(* RESETS AXES IF PHASE DONE AND CONNECTION DONE AND DISABLED *)
IF 	phase_done
	AND connection_done
	AND axis_is_disabled(axis)
THEN
	phase_done := FALSE;
	connection_done := FALSE;
END_IF

(* CLEARS PHASE AND CONNECTION ERRORS ON STOP *)
IF 	machine_is_stopped(csp.mch)
	OR machine_is_stop_emergency_active(csp.mch)
THEN
	phase_error := FALSE;
	connection_error := FALSE;	
END_IF

(* Overflow protection of engage count *)
IF	engage_count > 32000
THEN
	engage_count := 0;
END_IF

phase();

connection();

_handle_messages();

_write_output();

ACTION _handle_messages:
;
END_ACTION

ACTION _handle_process_test:
;
END_ACTION

ACTION _mode_manager:
IF process_mode_req_is_pending(prc)
THEN
    process_apply_mode_req_first_step(prc);
    CASE process_get_mode(prc) OF
        MODE_TO_ABSENT:
			;
        MODE_TO_INACTIVE:
			;
        MODE_TO_TEST:
			;
        MODE_TO_OPERATIONAL:
			;
    END_CASE
    process_apply_mode_req_second_step(prc);
END_IF
END_ACTION

ACTION _object_manager:
IF objects_initialization()
THEN
	sub_process_init(
		object_name					:= 'csp_case_virtualMaster.prc', 
		process						:= csp_case.prc, 
		CONVERSION_this				:= prc);
		
	prc_path 						:= process_get_path(prc);
	
	boolean_init(
        object_name:= CONCAT(prc_path, 'Axis_faulted'),
        process:= prc,
        CONVERSION_this:= Axis_faulted);
		
	axis_init(
		object_name								:= CONCAT(prc_path, '_axis'), 
		axis_type								:= AXIS_TYPE_VIRTUAL, 
		encoder_scaling_factor					:= G_VIRTUAL_ENCODER_SCALING_FACTOR_DEGPINC,
		modulo									:= G_MODULO_360_DEG, 
		process									:= prc, 
		CONVERSION_this							:= axis);
	
	axis_set_max_dynamic(
		reference_velocity						:=	MOTOR_MAX_VELOCITY_DEGPS,
		velocity								:=	MOTOR_MAX_VELOCITY_DEGPS,
		acceleration							:=	MOTOR_MAX_ACCELLERATION_DEGPS2,
		deceleration							:=	MOTOR_MAX_DECELLERATION_DEGPS2,
		jerk									:=	MOTOR_MAX_JERK_DEGPS3,
		following_error							:=	MOTOR_MAX_FOLLOWING_ERROR_DEG,
		CONVERSION_this							:=	axis);
	
	jog_manager_add_axis(
		list_index					:= JOG_LIST_CSP_CASE_VIRTUAL,
		axis						:= axis,
		master_axis					:= TRUE,
		jog_type					:= JOG_TYPE_ROTATIVE_PLUS,
		sw_limit_positive			:= 0.0,
		sw_limit_negative			:= 0.0,
		CONVERSION_this				:= csp_main_jogManager.jog_manager_virtual);

	
    digital_check_and_message_init(
        object_name:= CONCAT(prc_path, 'Axis_faulted_active_dchk'),
        alarm_if_input_off:= FALSE,
        alarm_delay:= 0,
        enabled_at_powerup:= TRUE,
        individual_reset:= FALSE,
        machine_reaction:=  MACHINE_REACTION_EMERGENCY_STOP,//MACHINE_REACTION_EMERGENCY_STOP,
        typology:=  MESSAGE_TYPOLOGY_ABNORMAL,//MESSAGE_TYPOLOGY_OBLIGATION,
        process:= prc,
        CONVERSION_this:= Axis_faulted_active_dchk);
       
       
    digital_check_add_boolean(
        boolean:= Axis_faulted,
        CONVERSION_this:= Axis_faulted_active_dchk);

		
	process_message_init(
		object_name					:=	CONCAT(prc_path, '_runout_complete'), 
		behaviour					:=	MESSAGE_BEHAVIOUR_EVENT,
		reset_timeout				:=	0,
		disableable					:=	TRUE,
		individual_reset			:=	FALSE,
		machine_reaction			:=	MACHINE_REACTION_STOP_IN_PHASE_ONE,
		typology					:=	MESSAGE_TYPOLOGY_ABNORMAL,
		process						:=	prc,
		CONVERSION_this				:=	runout_complete);
		
		
	process_message_init(
		object_name					:=	CONCAT(prc_path, '_phase_faulted_aem'), 
		behaviour					:=	MESSAGE_BEHAVIOUR_EVENT,
		reset_timeout				:=	0,
		disableable					:=	TRUE,
		individual_reset			:=	FALSE,
		machine_reaction			:=	MACHINE_REACTION_NORMAL_STOP,
		typology					:=	MESSAGE_TYPOLOGY_ABNORMAL,
		process						:=	prc,
		CONVERSION_this				:=	phase_faulted_aem);
	
	timer_init(
		object_name					:= CONCAT(prc_path, 'phase_time_out_tmr'),
		process						:= prc,
		CONVERSION_this				:= phase_time_out_tmr);
		
	process_message_init(
		object_name					:=	CONCAT(prc_path, 'debug_immediate_stop_aem'), 
		behaviour					:=	MESSAGE_BEHAVIOUR_STATE,
		reset_timeout				:=	0,
		disableable					:=	TRUE,
		individual_reset			:=	FALSE,
		machine_reaction			:=	MACHINE_REACTION_NORMAL_STOP,
		typology					:=	MESSAGE_TYPOLOGY_ABNORMAL,
		process						:=	prc,
		CONVERSION_this				:=	debug_immediate_stop_aem);
		
	timer_init(
		object_name					:= CONCAT(prc_path, 'connection_time_out_tmr'),
		process						:= prc,
		CONVERSION_this				:= connection_time_out_tmr);
		
		
	process_message_init(
		object_name					:=	CONCAT(prc_path, '_connection_faulted_aem'), 
		behaviour					:=	MESSAGE_BEHAVIOUR_EVENT,
		reset_timeout				:=	0,
		disableable					:=	TRUE,
		individual_reset			:=	FALSE,
		machine_reaction			:=	MACHINE_REACTION_NORMAL_STOP,
		typology					:=	MESSAGE_TYPOLOGY_ABNORMAL,
		process						:=	prc,
		CONVERSION_this				:=	connection_faulted_aem);
		
	motorization_conditioner_init(
		object_name					:=	CONCAT(prc_path, 'connection_done_motcond'),
		velocity_limit				:=	0.0,
		velocity_limit_active		:=	FALSE,
		idle_handshake_active		:=	FALSE,
		execute_handshake_active	:=	TRUE,
		hold_handshake_active		:=	FALSE,
		suspend_handshake_active	:=	FALSE,
		complete_handshake_active	:=	FALSE,
		abort_handshake_active		:=	FALSE,
		stop_handshake_active		:=	FALSE,
		origin						:=	MOTORIZATION_CONDITIONER_ORIGIN_INTERNAL,
		manager						:=	csp_main_motorization_manager.motm,
		process						:=	prc,
		CONVERSION_this				:=	connection_done_motcond);
   
		
	phase_init(
        object_name 				:= CONCAT(prc_path, '_run_check_ph'),
        phase 						:= 0,	//Set at runtime!
        delay 						:= 0,
        max_compensation 			:= 0,
        generator 					:= csp_main_motorization_virtualManager.phgen,
        process 					:= prc,
        CONVERSION_this 			:= run_check_ph);	
		
	phase_init(
        object_name 				:= CONCAT(prc_path, '_load_check_ph_jog'),
        phase 						:= 0,	//Set at runtime!
        delay 						:= 0,
        max_compensation 			:= 0,
        generator 					:= csp_main_motorization_virtualManager.phgen,
        process 					:= prc,
        CONVERSION_this 			:= load_check_ph_jog);	
		

END_IF

IF objects_running()
THEN
	process_cycle(prc);
	motorization_conditioner_cycle(connection_done_motcond);
	
	phase_cycle(run_check_ph);
	phase_cycle(load_check_ph_jog);
	axis_cycle(axis);
	digital_check_cycle(Axis_faulted_active_dchk);
END_IF
END_ACTION

ACTION _read_process_image:
;
END_ACTION

ACTION _read_var_input:
disable_req := csp_case.disable_req;
END_ACTION

ACTION _set_runtime_properties:
(* Cam management *)
IF 	connection_done
THEN
	active_cam := axis.engaged_cam.cam_id;
END_IF

(******************** DEBUG *****************************)

IF 
( (* USED FOR PRIMING THE CASE SIDE WITH A CASE SO IT IS READY TO LOAD IMMEDIATELY FROM TRANSFER *)
	(
		NOT csp_case_loader.cases_primed 
		AND 
			(
				NOT csp_case_loader.case_at_loader
				OR
				(
					csp_case_loader.case_at_loader
					AND csp_transfer_upstacker.stack_in_case_at_loader
				)
					
			)
	)
	AND NOT csp_case_transport_virtualMaster.stop_for_reject
	AND axis_is_cam_engaged(csp_case_feed_virtualMaster.axis)
	AND NOT message_is_on(csp_case_discharge_reject_sensors.downstream_backup_di_dchk.alarm_asm.message)
	AND NOT message_is_on(csp_main_interface.Cartoner_Stop_Request_aem)
	AND NOT motorization_manager_is_held(csp_main_motorization_manager.motm)//message_is_on(csp_main_interface.Cartoner_Stop_Request_aem)
	//AND NOT csp_case_feed_magazine.suspend_request_aml_zone	
)
THEN
	condition1 := TRUE;
ELSE
	condition1 := FALSE;
END_IF

IF
( (* STACK IS READY AND WAITING ON TRANSFER TO RUN (CASE & LOAD AT LOAD SR STEP AND CASE AT FEED SR STEP)*)
	csp_case_loader.case_at_loader
	AND csp_transfer_upstacker.stack_in_case_at_loader
	AND csp_case_loader.cases_primed 
	AND csp_case_fc_ls_upper_leadingMinorCloser.at_upstream_pos
	AND NOT csp_case_transport_virtualMaster.stop_for_reject
	AND axis_is_cam_engaged(csp_case_feed_virtualMaster.axis)
	AND axis_is_cam_engaged(csp_case_transport_virtualMaster.axis)
	AND NOT message_is_on(csp_case_discharge_reject_sensors.downstream_backup_di_dchk.alarm_asm.message)
	AND NOT message_is_on(csp_main_interface.Cartoner_Stop_Request_aem)
	AND NOT motorization_manager_is_held(csp_main_motorization_manager.motm)
	//AND NOT csp_case_feed_magazine.suspend_request_aml_zone	
)
THEN
	condition2 := TRUE;
ELSE
	condition2 := FALSE;
END_IF

IF 
( (* STACK IS READY AND WAITING ON TRANSFER TO RUN (NO CASE & LOAD AT LOAD SR STEP AND CASE AT FEED SR STEP) *)
	NOT csp_case_loader.case_at_loader
	AND NOT csp_transfer_upstacker.stack_in_case_at_loader
	AND csp_case_loader.cases_primed 
	//AND NOT csp_case_fc_ls_upper_leadingMinorCloser.at_upstream_pos  //removed because no case at loader
	AND NOT csp_case_transport_virtualMaster.stop_for_reject
	AND axis_is_cam_engaged(csp_case_feed_virtualMaster.axis)
	AND axis_is_cam_engaged(csp_case_transport_virtualMaster.axis)
	AND NOT message_is_on(csp_case_discharge_reject_sensors.downstream_backup_di_dchk.alarm_asm.message)
	AND NOT message_is_on(csp_main_interface.Cartoner_Stop_Request_aem)
	AND NOT motorization_manager_is_held(csp_main_motorization_manager.motm)//message_is_on(csp_main_interface.Cartoner_Stop_Request_aem)
	//AND NOT csp_case_feed_magazine.suspend_request_aml_zone	
	)
THEN
	condition3 := TRUE;
ELSE
	condition3 := FALSE;
END_IF
END_ACTION

ACTION _write_output:
;
END_ACTION

ACTION connection:
connection_conditions :=	
	NOT process_message_is_on(connection_faulted_aem)
	//AND
	//NOT jog_manager_is_jog_axis_active(JOG_LIST_CSP_CASE_VIRTUAL, csp_main_jogManager.jog_manager_virtual)
	AND
	phase_done;

(* connection_done reset *)
IF	connection_done
	AND	
	NOT connection_conditions
	AND
	NOT csp.o_machine_is_running
THEN
	connection_done := FALSE;
END_IF

(* Exit conditions *)
IF	NOT connection_conditions 
	AND
	NOT motorization_manager_is_stopping(csp_main_motorization_manager.motm)	
THEN	
	connection_status_next := CSP_CASE_STATUS_CONNECTION_ERROR;
	connection_status := connection_status_next;	
END_IF

(*************** MACHINE STATUS ***************)
CASE connection_status OF

	CSP_CASE_STATUS_CONNECTION_START:	(* Start connection *)
		IF	(
				motorization_manager_is_starting(csp_main_motorization_manager.motm) //TODOPZ: da decidere a che livello usare le variabili di i e o: wn_feeding.i_motorization_is_starting?					
				//AND axis_is_cam_engaged(csp_case_feed_virtualMaster.axis)
				//AND axis_is_cam_engaged(csp_case_glue_virtualMaster.axis)
				AND 
					(
						axis_is_cam_engaged(csp_case_transport_virtualMaster.axis) 
						OR 
						csp_case_transport_virtualMaster.stop_for_reject
					)
				//AND axis_is_cam_engaged(csp_case_loader_virtualMaster.axis)
				//OR
				//jog_manager_is_jog_axis_active(JOG_LIST_CSP_CASE_VIRTUAL, csp_main_jogManager.jog_manager_virtual)
			)
			THEN
				connection_running := TRUE;
				connection_status_next := CSP_CASE_STATUS_CONNECTION_ENGAGE;
		END_IF
		
	CSP_CASE_STATUS_CONNECTION_ENGAGE:		
	
		master_offset_phase := csp_main_motorization_virtualManager.axis.actual_modulo_position;		
	
		axis_engage_cam(
			cam_id							:=	active_cam,	
			master_engage_mode				:=	AXIS_CAM_ENGAGE_RELATIVE,
			slave_engage_mode				:=	AXIS_CAM_ENGAGE_RELATIVE,
			activation_mode					:=	AXIS_CAM_ACTIVATION_IMMEDIATELY,
			activation_position				:=	0.0,
			master_scaling_mode				:=	AXIS_CAM_SCALING_MODE_USER_DEFINED,
			slave_scaling_mode				:=	AXIS_CAM_SCALING_MODE_AUTOOFFSET,
			master_offset					:=	LMOD(home_position_master_offset_deg + master_offset_phase, axis_get_modulo(csp_main_motorization_virtualManager.axis)),
			slave_offset					:=	0.0,
			master_scaling					:=	master_scaling,
			slave_scaling					:=	slave_scaling,
			interpolation_type				:=	AXIS_CAM_INTERPOLATION_SPLINE,	 
			master							:=	csp_main_motorization_virtualManager.axis,
			CONVERSION_this					:=	axis);
		
		connection_status_next:= CSP_CASE_STATUS_CONNECTION_ENGAGED;
	
	CSP_CASE_STATUS_CONNECTION_ENGAGED:
	
		IF active_cam = 0
		THEN
			active_cam := next_cam;
		END_IF
	
		IF 	axis_is_cam_engaged(axis) 
		THEN				
			IF	active_cam <> next_cam
			THEN							
				connection_status_next := CSP_CASE_STATUS_CONNECTION_CHANGE_CAM;
			ELSE
				connection_status_next:= CSP_CASE_STATUS_CONNECTION_DONE;
			END_IF
		END_IF
		
	CSP_CASE_STATUS_CONNECTION_CHECK_CHANGE_CAM:	
					
		IF 	dwell
		THEN
			next_cam := DWELL_CAM;
			dwell:= FALSE;	
		END_IF
				
		IF 	run
		THEN
			next_cam := FORWARD_CAM;
			run := FALSE;
		END_IF	
		
		IF	(active_cam <> next_cam)
			AND 
			connection_conditions
		THEN							
			connection_status_next := CSP_CASE_STATUS_CONNECTION_CHANGE_CAM;
		END_IF
			
		//IF	NOT connection_motorization_moving
		//THEN
			//connection_status_next := CSP_CASE_STATUS_CONNECTION_DONE;
		//END_IF
	
	CSP_CASE_STATUS_CONNECTION_CHANGE_CAM:	
		engage_count := engage_count + 1;

		axis_engage_cam(
			cam_id							:=	next_cam,	
			master_engage_mode				:=	AXIS_CAM_ENGAGE_RELATIVE,
			slave_engage_mode				:=	AXIS_CAM_ENGAGE_RELATIVE,
			activation_mode					:=	AXIS_CAM_ACTIVATION_NEXT_CYCLE,
			activation_position				:=	0,
			master_scaling_mode				:=	AXIS_CAM_SCALING_MODE_USER_DEFINED,
			slave_scaling_mode				:=	AXIS_CAM_SCALING_MODE_USER_DEFINED,
			master_offset					:=	home_position_master_offset_deg, 
			slave_offset					:=	0.0,
			master_scaling					:=	master_scaling,
			slave_scaling					:=	slave_scaling,
			interpolation_type				:=	AXIS_CAM_INTERPOLATION_SPLINE,	 
			master							:=	csp_main_motorization_virtualManager.axis,
			CONVERSION_this					:=	axis);	
	
		IF	motorization_manager_is_starting(csp_main_motorization_manager.motm)
		THEN
			connection_status_next := CSP_CASE_STATUS_CONNECTION_DONE;
		ELSE
			//IF axis_is_cam_engaged(axis)
			//THEN
			connection_status_next := CSP_CASE_STATUS_CONNECTION_WAIT_NEW_CAM;
		END_IF
		//END_IF
	
	CSP_CASE_STATUS_CONNECTION_WAIT_NEW_CAM:
	
		IF	NOT connection_motorization_moving
		THEN
			connection_status_next := CSP_CASE_STATUS_CONNECTION_DONE;
		END_IF
	
		IF	active_cam = next_cam
		THEN
			connection_status_next := CSP_CASE_STATUS_CONNECTION_CHECK_CHANGE_CAM;
		END_IF
		
	CSP_CASE_STATUS_CONNECTION_DONE:	(* Connection done *)	
	
		connection_running := FALSE;
		connection_done := TRUE;
		
		IF	motorization_manager_is_starting(csp_main_motorization_manager.motm)
		THEN
			motorization_conditioner_start_done(connection_done_motcond);							
			//IF	active_cam <> next_cam
			//THEN
				//connection_status_next := CSP_CASE_STATUS_CONNECTION_WAIT_NEW_CAM;
			//ELSE
				
			//END_IF
		END_IF
		
		IF csp.o_machine_is_running 
		THEN
			connection_status_next := CSP_CASE_STATUS_CONNECTION_CHECK_CHANGE_CAM;
		ELSE
			;//DO NOTHING!! NO NEED TO RUN WHILE NOT IN EXECUTE
		END_IF
	
	CSP_CASE_STATUS_CONNECTION_ERROR:	(* Connection error *)	
	
		IF 	connection_running
		THEN
			axis_disable(axis);
			connection_error := TRUE;						
		END_IF
		connection_running	:= FALSE;
		connection_done 	:= FALSE;	
		
		IF	connection_conditions
		THEN		
			connection_status_next := CSP_CASE_STATUS_CONNECTION_START;
		END_IF
		
END_CASE

IF 	NOT debug_state_machine
	OR
	debug_connection_machine_one_step	
THEN
	connection_status := connection_status_next;
	debug_connection_machine_one_step := FALSE;
END_IF

connection_motorization_moving	:= 
	motorization_manager_is_starting(csp_main_motorization_manager.motm)
	OR
	motorization_manager_is_execute(csp_main_motorization_manager.motm)
	OR
	motorization_manager_is_stopping(csp_main_motorization_manager.motm)
	OR
	motorization_manager_is_suspended(csp_main_motorization_manager.motm)
	OR
	motorization_manager_is_suspending(csp_main_motorization_manager.motm)
	OR
	motorization_manager_is_unsuspending(csp_main_motorization_manager.motm)
	OR 
	motorization_manager_is_holding(csp_main_motorization_manager.motm)
	OR
	motorization_manager_is_held(csp_main_motorization_manager.motm)
	OR
	motorization_manager_is_unholding(csp_main_motorization_manager.motm);	
	
(* Connection timeout *)
IF	(connection_running
	AND NOT debug_state_machine)	
	OR connection_error
THEN
	IF	timer_is_expired(connection_time_out_tmr)
	THEN
		process_message_set(1, connection_status, 0, connection_faulted_aem);
	END_IF
ELSE
	timer_restart(10000, connection_time_out_tmr);
END_IF
END_ACTION

ACTION phase:
phase_conditions :=
	axis_is_ok(FALSE, axis)
	AND
	process_is_ready(prc)
	AND
	process_subtree_is_ready(prc)
	AND
	NOT jog_manager_is_jog_axis_active(JOG_LIST_CSP_CASE_VIRTUAL, csp_main_jogManager.jog_manager_virtual)
	AND
	csp_main_motorization.motorization_axis_redefined_at_powerup
	AND
	NOT disable_req;		
	
(* phase_done reset *)
IF	phase_done
	AND
	NOT phase_conditions
	//AND 
	//NOT csp.o_machine_is_running
THEN
	//axis_disable(axis);
	phase_done:= FALSE;
END_IF

(* Exit condition *)
IF 	NOT phase_conditions
THEN
	phase_status_next := CSP_CASE_PHASE_STATUS_ERROR;
	phase_status := phase_status_next;	
END_IF

(*************** MACHINE STATUS ***************)
CASE phase_status OF

	CSP_CASE_PHASE_STATUS_START:	(* Start phasing *)
	
		IF	(
				motorization_manager_is_starting(csp_main_motorization_manager.motm) //TODOPZ: da decidere a che livello usare le variabili di i e o: wn_feeding.i_motorization_is_starting?					
				//OR
				//jog_manager_is_jog_axis_active(JOG_LIST_CSP_CASE_VIRTUAL, csp_main_jogManager.jog_manager_virtual)
			)
		THEN
			phase_running := TRUE;			
			phase_status_next := CSP_CASE_PHASE_STATUS_DISABLE;
		END_IF
						
	CSP_CASE_PHASE_STATUS_DISABLE:
	
		axis_disable(axis);		
		
		IF 	axis_is_disabled(axis)
		THEN
			phase_status_next := CSP_CASE_PHASE_STATUS_ENABLE;
		END_IF
		
	CSP_CASE_PHASE_STATUS_ENABLE:
	
		axis_enable(axis);
		
		IF 	axis_is_enabled(axis)
		THEN
			phase_status_next := CSP_CASE_PHASE_STATUS_ENABLED;
		END_IF
		
	CSP_CASE_PHASE_STATUS_ENABLED:
	
		IF 	axis_is_standstill(axis) 
		THEN
			phase_status_next := CSP_CASE_PHASE_STATUS_CALCULATE_SLAVE_POSITION_REQUEST;								
		END_IF
		
	CSP_CASE_PHASE_STATUS_CALCULATE_SLAVE_POSITION_REQUEST:
	
		slave_position_has_been_calculated := FALSE;
	
		(* Gets the position of the master axis *)
		axis_calculate_cam_slave_master_position_deg := 
			LMOD(axis_get_actual_modulo_position(csp_main_motorization_virtualManager.axis)
			+ home_position_master_offset_deg, G_MODULO_360_DEG);
			
		(* Gets cam data for slave axis to master *)
		IF 	axis_calculate_cam_slave_dynamics_data(
				cam_id := active_cam,
				master_scaling := master_scaling,
				master_position := axis_calculate_cam_slave_master_position_deg,
				slave_scaling := slave_scaling,
				CONVERSION_this := axis)
		THEN
			phase_status_next := CSP_CASE_PHASE_STATUS_CALCULATING_SLAVE_POSITION;
		END_IF
	
	CSP_CASE_PHASE_STATUS_CALCULATING_SLAVE_POSITION:
	
		IF 	axis_cam_slave_dynamics_data_calculated(axis)
		THEN
			axis_calculated_cam_slave_position_deg := axis_get_cam_slave_dynamics_position(axis);
			slave_position_has_been_calculated := TRUE;
			phase_status_next := CSP_CASE_PHASE_STATUS_REQUEST;
		END_IF
		
	CSP_CASE_PHASE_STATUS_REQUEST:
		
		IF	axis_is_standstill(axis)
		THEN
		 	axis_move_absolute(
				position 		:= axis_calculated_cam_slave_position_deg,
				velocity 		:= phase_velocity_degps,
				direction		:= AXIS_SHORTEST_WAY,
				acceleration 	:= MOTOR_MAX_ACCELLERATION_DEGPS2,
				deceleration 	:= MOTOR_MAX_DECELLERATION_DEGPS2, 
				jerk 			:= MOTOR_MAX_JERK_DEGPS3, 
				buffer_mode 	:= AXIS_BUFFER_MODE_BUFFERED,
				CONVERSION_this := axis
				); 
			
		END_IF

		IF 	axis_is_absolute_moving(axis)
		THEN
			phase_status_next	:=	CSP_CASE_PHASE_STATUS_PHASING;
		END_IF

	CSP_CASE_PHASE_STATUS_PHASING:

		IF 	axis_is_standstill(axis)
		THEN
			phase_status_next	:=	CSP_TRANSFER_STATUS_PHASED;
		END_IF

	CSP_TRANSFER_STATUS_PHASED:

		IF 	engage_enable
		THEN
			phase_status_next := CSP_CASE_PHASE_STATUS_DONE;
		END_IF
		
		
	CSP_CASE_PHASE_STATUS_DONE:	(* Phase done *)		
	
		phase_running := FALSE;
		phase_done := TRUE;				
	
	CSP_CASE_PHASE_STATUS_ERROR:	(* Phase error *)
		

		IF	phase_running
		THEN
			phase_error := TRUE;
			axis_disable(axis);									
		END_IF
		phase_running := FALSE;
		
		IF	phase_conditions 	
		THEN
			phase_status_next := CSP_CASE_PHASE_STATUS_START;
		END_IF
		
END_CASE

IF 	NOT debug_state_machine
	OR
	debug_phase_machine_one_step	
THEN
	phase_status := phase_status_next;
	debug_phase_machine_one_step := FALSE;
END_IF

(* Phasing timeout *)
IF (phase_running
	AND NOT debug_state_machine)
	OR phase_error
THEN
	IF	timer_is_expired(phase_time_out_tmr)
	THEN
		process_message_set(1, phase_status, 0, phase_faulted_aem);
	END_IF
ELSE
	timer_restart(10000, phase_time_out_tmr);
END_IF
END_ACTION

END_PROGRAM

// ---- Application/CSP/Case/Loader/Pusher/csp_case_loader_pusher.TcPOU
(*********************************** G.D S.p.A. - Technical Department ***********************************
============= PROGRAM INFO ============
FOLDER:             TBD
MACHINES INVOLVED:  TBD 

============= DESCRIPTION =============
csp machine declaration

============= REVISIONS ===============
Date		Version	 	Author      	Description             
----------	-------		------------  	--------------------------------------------
2019/04/05 	0000.00	 	M.Grasso		Creation of the PRG

**********************************************************************************************************)
(*$R process_ref := prc; $*)
PROGRAM csp_case_loader_pusher
VAR
	
	prc:											process;
	prc_path:										STRING;
	
	axis:											axis;
	
	fsm_next_status: 								CSP_CASE_LOADER_STATUS_ENUM;
	axis_calculate_cam_slave_master_position_deg: 	LREAL;
	axis_calculated_cam_slave_position_deg: 		LREAL;
	cam_id:											INT := CASE_LOADER_PUSHER_RUN_CAM;
	slave_scaling:									LREAL := 807; (*$P $*) //orginally 360
	master_scaling:									LREAL := 1; 
	master_offset:									LREAL := 240;(*$P $*)
	slave_offset: 									LREAL := 0;
	debug_state_machine: 							BOOL :=FALSE;
	debug_state_machine_one_step: 					BOOL := FALSE;
	fsm_status: 									CSP_CASE_LOADER_STATUS_ENUM;
	phase_velocity_degps: 							LREAL := 50;
	slave_position_has_been_calculated: 			BOOL := FALSE;
	fsm_enable_condition: 							BOOL := FALSE;
	disable_req: 									BOOL := FALSE;
	phase_enable:									BOOL:=TRUE;
	torque_limit:									INT := 2000;    (*$P $*)
	torque_limit_old:								INT;
	
    in_accu_safe_pos:                               BOOL := FALSE;
    accu_tolerance:                                 LREAL := 5;
    accu_safe_pos:                                  LREAL := 0;	
	
	direction_FWD: 									BOOL;
	CAM_CHANGE_CHECK_DEG:							LREAL := 5;
	cam_change_check_ph:							phase;
	
	
	(* RFID *)
	rfid_check_pos:									LREAL := 0; (*$P $*)
	check_pls_tolerance:							LREAL := 2;
	rfid_value:										BYTE;
	rfid_value_to_write:							BYTE;
	
	rfid_input_buffer:								iol_slave_bis00lh_pdo_input;
	rfid_input_bitheader_1:							iol_slave_bis00lh_bitheader_input;
	rfid_input_bitheader_2:							iol_slave_bis00lh_bitheader_input;
			
	rfid_output_buffer:								iol_slave_bis00lh_pdo_output;
	rfid_output_bitheader_1:						iol_slave_bis00lh_bitheader_output;
	rfid_output_bitheader_2:						iol_slave_bis00lh_bitheader_output;
	
	RFID_read_write_status:							csp_case_loader_rfid_status_enum;
	RFID_read_write_status_next:					csp_case_loader_rfid_status_enum;
	RFID_read_write_debug:							BOOL := FALSE;
	RFID_read_write_one_step:						BOOL := FALSE;
	RFID_read_write_running:						BOOL;
	RFID_read_write_tmr:							timer;
	RFID_read_write_error_msg:						message;
	
	rfid_start_toggle:								BOOL := FALSE;
	rfid_shutdown_toggle:							BOOL := FALSE;
	rfid_write_toggle:								BOOL := FALSE;
	rfid_write_done:								BOOL := FALSE;
	rfid_read_toggle:								BOOL := FALSE;
	rfid_read_done:									BOOL := FALSE;

	servo_on_condition: 							BOOL;
	enable_delay: 									TON;
	Torque_force_constant: 							LREAL := 1.2;
	RisingEdgeRFIDSelect:							R_Trig;
END_VAR

VAR CONSTANT
	(*Just in case you prefer having constants instead of numbers*)
	MOTOR_MAX_VELOCITY_DEGPS:				LREAL := 9600;
	MOTOR_MAX_ACCELLERATION_DEGPS2:			LREAL := 4800;
	MOTOR_MAX_DECELLERATION_DEGPS2:			LREAL := 4800;
	MOTOR_MAX_JERK_DEGPS3:					LREAL := 100000000; 
	MOTOR_MAX_FOLLOWING_ERROR_DEG:			LREAL := 2;
END_VAR

_read_var_input();

_object_manager();

IF NOT objects_running()
THEN
	RETURN;	
END_IF

_read_process_image();

_mode_manager();

CASE process_get_mode(prc) OF
	MODE_ABSENT:
		IF axis_get_mode(axis) = MODE_TEST
		THEN
			safety_integrated_series_close(csp_case_main_safety_drives_SD8500.chA_smes_sis);
		END_IF
		RETURN;
	MODE_INACTIVE:
		RETURN;
	MODE_TEST:
		_handle_process_test();
END_CASE

_set_runtime_properties();

(********************************* BODY *********************************)
axis.actual_torque := (axis.actual_current * Torque_force_constant)/1000;

RisingEdgeRFIDSelect(
					CLK := (csp_main_accuChange.RFID_reader_list_accuchange = LOADER_PUSHER_READER) 
					);
				
IF RisingEdgeRFIDSelect.Q
THEN
	RFID_read_write_status := CSP_CASE_LOADER_RFID_STATUS_START;
END_IF

IF 	csp_main_accuChange.RFID_reader_list_accuchange = LOADER_PUSHER_READER
THEN
	RFID();
END_IF

(*FSM Control*)

phase_set_data(
	phase				:= CAM_CHANGE_CHECK_DEG,
	delay				:= 0,			
	max_compensation	:= 0,			
	CONVERSION_this		:= cam_change_check_ph);
	
	
(*disable_req *) //read_var_input
				
IF 	ABS(axis.actual_position - accu_safe_pos)  < accu_tolerance
THEN
	in_accu_safe_pos := TRUE;
ELSE
	in_accu_safe_pos := FALSE;   
END_IF		

(* VERIFIES LOADER IS CLEAR AND WILL NOT RUN *)
		
				
fsm_enable_condition := axis_is_ok(FALSE, axis)
						AND
						process_is_ready(prc)
						AND
						process_subtree_is_ready(prc)
						AND
						servo_on_condition
						AND						
						(csp_main_motorization.motorization_axis_redefined_at_powerup OR csp_main_accuchange.Brand_Change_Occurred)
						//AND
						//NOT jog_manager_is_jog_axis_active(SMTR8503_CASE_LOADER_PUSHER, csp_main_jogManager.jog_manager_real)
						AND
						NOT disable_req;

IF	NOT fsm_enable_condition
	AND
	fsm_status <> CSP_CASE_LOADER_STATUS_DISABLED
	AND
	fsm_status < CSP_CASE_LOADER_STATUS_STOP_REQUEST
THEN
	fsm_status	:=	CSP_CASE_LOADER_STATUS_DISABLE_REQUEST;
END_IF;

IF torque_limit <> Torque_limit_old
	THEN
	IF soe_drive_channel_write_parameter(
		channel:=csp_case_loader_pusher.axis.soe_drive_channel, 
		idn:= S_0_IDN + 92, 
		data_element:=soe_drive_element_value , 
		data_source:= ADR(torque_limit), 
		data_lenght:= SIZEOF(torque_limit), 
		CONVERSION_this:= csp_case_loader_pusher.axis.soe_drive^)= SOE_DRIVE_RETURN_VALUE_DONE 
		THEN
		torque_limit_old := Torque_limit;
	END_IF	
END_IF
	
CASE fsm_status OF
	
	CSP_CASE_LOADER_STATUS_NOT_INITIALIZED:
	
        IF	axis_is_ok(return_when_absent := TRUE, CONVERSION_this := axis)
        THEN
            fsm_next_status := CSP_CASE_LOADER_STATUS_DISABLED;
        END_IF

	CSP_CASE_LOADER_STATUS_DISABLED:

		IF	fsm_enable_condition
			AND
			(
				(motorization_manager_is_starting(csp_main_motorization_manager.motm))
				OR
				jog_manager_is_jog_axis_active(JOG_LIST_CSP_CASE_LOADER_VIRTUAL, csp_main_jogManager.jog_manager_virtual)
				//OR
				//jog_manager_is_jog_axis_active(JOG_LIST_CSP_CASE_VIRTUAL, csp_main_jogManager.jog_manager_virtual)	
			)
		THEN
			debug_state_machine := FALSE;
			fsm_next_status := CSP_CASE_LOADER_STATUS_ENABLE_REQUEST;
		END_IF;

	CSP_CASE_LOADER_STATUS_ENABLE_REQUEST:
	
		axis_enable(axis);
		IF axis_is_standstill(axis)
		THEN
			fsm_next_status	:=	CSP_CASE_LOADER_STATUS_ENABLED;
		END_IF;		

	CSP_CASE_LOADER_STATUS_ENABLED:

		IF 	NOT csp_main_accuChange.machine_size_complete
		THEN
			fsm_next_status	:= CSP_CASE_LOADER_STATUS_CHANGE_OVER_MODE;
		ELSE	
			fsm_next_status	:=	CSP_CASE_LOADER_STATUS_HOME_REQUEST;
		END_IF
		

	CSP_CASE_LOADER_STATUS_CHANGE_OVER_MODE:
		
		IF 	NOT in_accu_safe_pos
		THEN
			fsm_next_status	:=	CSP_CASE_LOADER_STATUS_ENABLE_CROSSPUSHERS;			
		END_IF;		
				

	CSP_CASE_LOADER_STATUS_ENABLE_CROSSPUSHERS:
	
		axis_enable(csp_transfer_crosspusher_horizontal.axis);
		axis_enable(csp_transfer_crosspusher_follower.axis);
		IF 	axis_is_enabled(csp_transfer_crosspusher_horizontal.axis)
			AND
			axis_is_enabled(csp_transfer_crosspusher_follower.axis)
		THEN
			fsm_next_status := CSP_CASE_LOADER_STATUS_MOVE_CROSSPUSHERS;
		END_IF

	
	CSP_CASE_LOADER_STATUS_MOVE_CROSSPUSHERS:
		
		IF 	axis_is_standstill(csp_transfer_crosspusher_horizontal.axis)
			AND
			axis_is_standstill(csp_transfer_crosspusher_follower.axis)
		THEN
			axis_move_absolute(
				position 		:= csp_transfer_crosspusher_horizontal.load_position,
				velocity 		:= phase_velocity_degps,
				direction		:= AXIS_SHORTEST_WAY,
				acceleration 	:= MOTOR_MAX_ACCELLERATION_DEGPS2,
				deceleration 	:= MOTOR_MAX_DECELLERATION_DEGPS2, 
				jerk 			:= MOTOR_MAX_JERK_DEGPS3, 
				buffer_mode 	:= AXIS_BUFFER_MODE_BUFFERED,
				CONVERSION_this := csp_transfer_crosspusher_horizontal.axis
				); 
				
			axis_move_absolute(
				position 		:= 500,
				velocity 		:= phase_velocity_degps,
				direction		:= AXIS_SHORTEST_WAY,
				acceleration 	:= MOTOR_MAX_ACCELLERATION_DEGPS2,
				deceleration 	:= MOTOR_MAX_DECELLERATION_DEGPS2, 
				jerk 			:= MOTOR_MAX_JERK_DEGPS3, 
				buffer_mode 	:= AXIS_BUFFER_MODE_BUFFERED,
				CONVERSION_this := csp_transfer_crosspusher_follower.axis
				); 
		END_IF
			
		IF	axis_is_absolute_moving(csp_transfer_crosspusher_follower.axis) 
			OR
			axis_is_absolute_moving(csp_transfer_crosspusher_horizontal.axis) 
		THEN
			fsm_next_status := CSP_CASE_LOADER_STATUS_VERIFY_CROSSPUSHERS_CLEAR;
		END_IF
		
	CSP_CASE_LOADER_STATUS_VERIFY_CROSSPUSHERS_CLEAR:
	
		IF 	csp_transfer_crosspusher_horizontal.axis.actual_position >= csp_transfer_crosspusher_horizontal.load_position
			AND csp_transfer_crosspusher_follower.axis.actual_position >= (csp_transfer_crosspusher_follower.slave_scaling-1)
			OR
			(
				rfid_input_bitheader_1.CP 
				AND rfid_input_bitheader_2.CP
			)
		THEN
			fsm_next_status := CSP_CASE_LOADER_STATUS_MOVE_AXIS_TO_POS;
		END_IF
	
		
	CSP_CASE_LOADER_STATUS_MOVE_AXIS_TO_POS:

		
		IF 	axis_is_standstill(axis)
			AND
			axis_is_standstill(csp_transfer_crosspusher_horizontal.axis)
			AND
			axis_is_standstill(csp_transfer_crosspusher_follower.axis)
		THEN
			axis_move_absolute(
				position 		:= accu_safe_pos,
				velocity 		:= motorization_manager_get_nominal_velocity(csp_main_motorization_manager.motm)*6,
				direction		:= AXIS_SHORTEST_WAY,
				acceleration 	:= MOTOR_MAX_ACCELLERATION_DEGPS2,
				deceleration 	:= MOTOR_MAX_DECELLERATION_DEGPS2,
				jerk 			:= MOTOR_MAX_JERK_DEGPS3, 
				buffer_mode 	:= AXIS_BUFFER_MODE_BUFFERED,
				CONVERSION_this := axis); 
		END_IF
	
		IF 	csp_main_accuChange.Motion_Motors_New_Size_Req
		THEN
			fsm_next_status	:=	CSP_CASE_LOADER_STATUS_HOME_REQUEST;
		END_IF;
		

	CSP_CASE_LOADER_STATUS_HOME_REQUEST: 

		fsm_next_status	:=	CSP_CASE_LOADER_STATUS_HOME_DONE;

	CSP_CASE_LOADER_STATUS_HOMING:

		axis.home.done := TRUE;

		IF 	axis_home_done(axis)
		THEN
			fsm_next_status	:=	CSP_CASE_LOADER_STATUS_HOME_DONE;
		END_IF

	CSP_CASE_LOADER_STATUS_HOME_DONE:
	
		IF 	phase_enable
			THEN
			fsm_next_status	:= CSP_CASE_LOADER_STATUS_CALCULATE_SLAVE_POSITION_REQUEST;
		END_IF
		
	CSP_CASE_LOADER_STATUS_CALCULATE_SLAVE_POSITION_REQUEST:
		
		(*Calculate a desired master axis position.
		Function used  LMOD: Ex. LMOD(400.56, 360) = 40.56
		home_position_master_offset_deg is helpful for changing the 1st term of LMOD*)
		
		axis_calculate_cam_slave_master_position_deg := 
		LMOD	(axis_get_actual_modulo_position(csp_case_loader_virtualMaster.axis) (*master axis*)
							+
				master_offset, (*initialized at 0° position*)
					G_MODULO_360_DEG											);
		(*master_scaling and slave_scaling initialized at 360° since the cams are normed in a range equal to 0-1.*)
		
			IF axis_calculate_cam_slave_dynamics_data(
					cam_id := cam_id,
					master_scaling := master_scaling,
					master_position := axis_calculate_cam_slave_master_position_deg,
					slave_scaling := slave_scaling,
					CONVERSION_this := axis)
			THEN
				fsm_next_status := CSP_CASE_LOADER_STATUS_CALCULATING_SLAVE_POSITION;
			END_IF

	CSP_CASE_LOADER_STATUS_CALCULATING_SLAVE_POSITION:
	
		IF	axis_cam_slave_dynamics_data_calculated(axis)
		THEN
		(*The “axis_get_cam_slave_dynamics_position” method returns the position of the slave within the cam plate table at the master position calculated for the instance specified: *)
			axis_calculated_cam_slave_position_deg :=(axis_get_cam_slave_dynamics_position(axis)+ slave_offset);
			slave_position_has_been_calculated := TRUE;
			
			IF 	axis.actual_position > axis_calculated_cam_slave_position_deg
			THEN 
				direction_FWD := FALSE;	// backward
			ELSIF axis.actual_position < axis_calculated_cam_slave_position_deg
			THEN
				direction_FWD := TRUE; //forward
			END_IF
	
			fsm_next_status := CSP_CASE_LOADER_STATUS_PHASE_REQUEST;
		END_IF


	CSP_CASE_LOADER_STATUS_PHASE_REQUEST:

		IF	axis_is_standstill(axis)
			AND csp_case_loader.follower_clear (* FOLLOWER IS CLEAR MEANING IT IS AT LOAD POSITION *)
			AND csp_case_loader.horizontal_clear (* HORIZONTAL IS CLEAR MEANING AT LOAD OR IN DIRECTION OF UPSTACK *)
		THEN

			axis_move_absolute(
				position 		:= axis_calculated_cam_slave_position_deg,(*calculated above, the slave is moved*)
				velocity 		:= phase_velocity_degps/2,
				direction		:= SEL(direction_FWD, AXIS_NEGATIVE_DIRECTION, AXIS_POSITIVE_DIRECTION),
				acceleration 	:= MOTOR_MAX_ACCELLERATION_DEGPS2,
				deceleration 	:= MOTOR_MAX_DECELLERATION_DEGPS2,
				jerk 			:= MOTOR_MAX_JERK_DEGPS3, 
				buffer_mode 	:= AXIS_BUFFER_MODE_BUFFERED,
				CONVERSION_this 			:= axis
				); 
			
		END_IF

		IF 	axis_is_absolute_moving(axis)
		THEN
			fsm_next_status	:=	CSP_CASE_LOADER_STATUS_PHASING;
		END_IF

	CSP_CASE_LOADER_STATUS_PHASING:

		IF 	axis_is_standstill(axis)
		THEN
			fsm_next_status	:=	CSP_CASE_LOADER_STATUS_PHASED;
		END_IF

	CSP_CASE_LOADER_STATUS_PHASED:

		fsm_next_status := CSP_CASE_LOADER_STATUS_CAM_ENGAGED_REQ;


	CSP_CASE_LOADER_STATUS_CAM_ENGAGED_REQ:

		axis_engage_cam(
			cam_id 			:= cam_id,
			master_engage_mode 	:= AXIS_CAM_ENGAGE_ABSOLUTE,
			slave_engage_mode 	:= AXIS_CAM_ENGAGE_ABSOLUTE, 
			activation_mode 	:= AXIS_CAM_ACTIVATION_IMMEDIATELY, 
			activation_position	:= 0,
			master_scaling_mode	:= AXIS_CAM_SCALING_MODE_USER_DEFINED,
			slave_scaling_mode	:= AXIS_CAM_SCALING_MODE_USER_DEFINED,
			master_offset 		:= master_offset,			//axis_calculate_cam_slave_master_position_deg, (*moved right  respect to the original Y axis of the cam profile*)
			slave_offset 		:= slave_offset,	//- axis_calculated_cam_slave_position_deg,  (*slave moved down of the same quantity already used in CSP_MACHINE_STATUS_PHASE_REQUEST via axis_move_absolute(..) *)
			master_scaling 		:= master_scaling,
			slave_scaling 		:= slave_scaling,
			interpolation_type 		:= AXIS_CAM_INTERPOLATION_SYSTEM_DEFAULT,
			master 			:= csp_case_loader_virtualMaster.axis,
			CONVERSION_this 	:= axis);		
	
		IF	axis_is_cam_engaged(axis)
		THEN
			fsm_next_status := CSP_CASE_LOADER_STATUS_CAM_ENGAGED;
		END_IF

	
	CSP_CASE_LOADER_STATUS_AXIS_ENGAGE_VERIFY :
		;
		
	CSP_CASE_LOADER_STATUS_CAM_ENGAGED:
	
		IF 	machine_is_stop_emergency_active(csp.mch)
			AND motorization_manager_is_stopped(csp_main_motorization_manager.motm)
		THEN
			fsm_next_status := CSP_CASE_LOADER_STATUS_DISENGAGE_REQUEST;
		END_IF
		
		IF 	phase_edge(cam_change_check_ph) (* CROSSPUSHER VIRTUAL AT CHECK PHASE DEG *)
			AND axis_is_cam_engaged(axis)
			AND NOT csp_case_loader.follower_clear
			AND NOT csp_case_loader.horizontal_clear
		THEN
			fsm_next_status := CSP_CASE_LOADER_STATUS_DISENGAGE_REQUEST;
		END_IF
		
	CSP_CASE_LOADER_STATUS_RUNNING:

		;
		
	CSP_CASE_LOADER_STATUS_DISENGAGE_REQUEST:

		fsm_next_status := CSP_CASE_LOADER_STATUS_DISENGAGING;
		
	CSP_CASE_LOADER_STATUS_DISENGAGING:
	
		IF 	axis_disengage(
				mode:= AXIS_DISENGAGE_AND_ON_PHASE_STOP, 
				position:= 0, 
				velocity:= 0, 
				acceleration:= MOTOR_MAX_ACCELLERATION_DEGPS2, 
				deceleration:= MOTOR_MAX_DECELLERATION_DEGPS2, 
				jerk:= MOTOR_MAX_JERK_DEGPS3, 
				CONVERSION_this:= axis)
		THEN
			fsm_next_status := CSP_CASE_LOADER_STATUS_CAM_ENGAGED_REQ;
		END_IF
	
	CSP_CASE_LOADER_STATUS_STOP_REQUEST:

		axis_stop(
		    deceleration 	:= MOTOR_MAX_DECELLERATION_DEGPS2,
		    jerk 			:= MOTOR_MAX_JERK_DEGPS3,
		    CONVERSION_this 			:= axis);

		IF 	axis_is_standstill(axis)
			OR
			NOT axis_is_ok(FALSE, axis)
			OR
			axis_is_disabled(axis)
		THEN
			fsm_next_status := CSP_CASE_LOADER_STATUS_DISABLE_REQUEST;
		END_IF

	CSP_CASE_LOADER_STATUS_DISABLE_REQUEST:
	
   		axis_disable(axis);
   		fsm_next_status := CSP_CASE_LOADER_STATUS_DISABLING;

	CSP_CASE_LOADER_STATUS_DISABLING:
	
        IF	axis_is_disabled(axis)
        THEN
            fsm_next_status := CSP_CASE_LOADER_STATUS_DISABLED;
        END_IF

END_CASE;

IF 	NOT debug_state_machine
	OR
	debug_state_machine_one_step
THEN
	fsm_status := fsm_next_status;
	debug_state_machine_one_step := FALSE;
END_IF
(************************************************************************)

_handle_messages();

_write_output();

ACTION _handle_messages:
;
END_ACTION

ACTION _handle_process_test:
;
END_ACTION

ACTION _mode_manager:
IF process_mode_req_is_pending(prc)
THEN
    process_apply_mode_req_first_step(prc);
    CASE process_get_mode(prc) OF
        MODE_TO_ABSENT:
			;
        MODE_TO_INACTIVE:
			;
        MODE_TO_TEST:
			;
        MODE_TO_OPERATIONAL:
			;
    END_CASE
    process_apply_mode_req_second_step(prc);
END_IF
END_ACTION

ACTION _object_manager:
IF objects_initialization()
THEN
	sub_process_init(
		object_name					:= 'csp_case_loader_pusher.prc', 
		process						:= csp_case_loader.prc, 
		CONVERSION_this				:= prc);
		
	prc_path 						:= process_get_path(prc);
	
(* axis smes *)
	IF csp_main_configurator.Physical_hw
	THEN
	
		axis_init(
			object_name								:= CONCAT(prc_path, '_axis'), 
			axis_type								:= AXIS_TYPE_SERVO, 
			encoder_scaling_factor					:= G_SERVO_ENCODER_SCALING_FACTOR_DEGPINC,
			modulo									:= G_NO_MODULO_DEG, 
			process									:= prc, 
			CONVERSION_this							:= axis);
			
		axis_add_safety_integrated_series(
			safety_integrated_series 	:= csp_case_main_safety_drives_SD8500.chA_smes_sis,
			CONVERSION_this				:= axis);
			
		axis_init_absolute_encoder_preset(
			position                                := 0.0,
			CONVERSION_this                         := axis);
			
	ELSE
		axis_init(
			object_name								:= CONCAT(prc_path, '_axis'), 
			axis_type								:= AXIS_TYPE_VIRTUAL, 
			encoder_scaling_factor					:= G_VIRTUAL_ENCODER_SCALING_FACTOR_DEGPINC,
			modulo									:= G_MODULO_1080_DEG, 
			process									:= prc, 
			CONVERSION_this							:= axis);		
				
	END_IF
	
	axis_set_max_dynamic(
		reference_velocity						:=	MOTOR_MAX_VELOCITY_DEGPS,
		velocity								:=	MOTOR_MAX_VELOCITY_DEGPS,
		acceleration							:=	MOTOR_MAX_ACCELLERATION_DEGPS2,
		deceleration							:=	MOTOR_MAX_DECELLERATION_DEGPS2,
		jerk									:=	MOTOR_MAX_JERK_DEGPS3,
		following_error							:=	MOTOR_MAX_FOLLOWING_ERROR_DEG,
		CONVERSION_this							:=	axis);
		
	axis_add_soe_drive(
		channel									:=	SOE_DRIVE_CHANNEL_A,
		soe_drive								:=	csp_case_main_drives.SD8500_drv,
		CONVERSION_this							:=	axis);
		
	jog_manager_add_axis(
		list_index								:= SMTR8503_CASE_LOADER_PUSHER,
		axis									:= axis,
		master_axis								:= FALSE,
		jog_type								:= JOG_TYPE_LINEAR,
		sw_limit_positive						:= 800,
		sw_limit_negative						:= 0,
		CONVERSION_this							:= csp_main_jogManager.jog_manager_real);
		
	process_message_init(
        object_name:= CONCAT(prc_path, '_RFID_read_write_error_msg'),
        behaviour:= MESSAGE_BEHAVIOUR_STATE,
        reset_timeout:= 0,
        disableable:= TRUE,
        individual_reset:= FALSE,
        machine_reaction:= MACHINE_REACTION_NO_STOP, //MACHINE_REACTION_STOP_IN_PHASE_ONE,
        typology:=  MESSAGE_TYPOLOGY_NOT_VISIBLE, //MESSAGE_TYPOLOGY_ABNORMAL,
        process:= prc,
        CONVERSION_this:= RFID_read_write_error_msg);
		
		
	phase_init(
        object_name 				:= CONCAT(prc_path, '_cam_change_check_ph'),
        phase 						:= 0,	//Set at runtime!
        delay 						:= 0,
        max_compensation 			:= 0,
        generator 					:= csp_case_transport_virtualMaster.transport_vm_phgen,
        process 					:= prc,
        CONVERSION_this 			:= cam_change_check_ph);	
		
END_IF

IF objects_running()
THEN
	phase_cycle(cam_change_check_ph);
	process_cycle(prc);
	axis_cycle(axis);
END_IF
END_ACTION

ACTION _read_process_image:
;
END_ACTION

ACTION _read_var_input:
disable_req := csp_case.disable_req;
;
END_ACTION

ACTION _set_runtime_properties:
enable_delay(IN:=axis_is_ready_to_enable(axis) , PT:=T#2S , Q=> servo_on_condition , ET=> );
END_ACTION

ACTION _write_output:
;
END_ACTION

ACTION RFID:
	(* RMH RFID TEST *)
rfid_input_bitheader_1.CP := rfid_input_buffer.ByteArr[0].0;
rfid_input_bitheader_1.AA := rfid_input_buffer.ByteArr[0].1;
rfid_input_bitheader_1.AE := rfid_input_buffer.ByteArr[0].2;
rfid_input_bitheader_1.AF := rfid_input_buffer.ByteArr[0].3;
rfid_input_bitheader_1.Bit4 := rfid_input_buffer.ByteArr[0].4;
rfid_input_bitheader_1._TO := rfid_input_buffer.ByteArr[0].5;
rfid_input_bitheader_1.HF := rfid_input_buffer.ByteArr[0].6;
rfid_input_bitheader_1.BB := rfid_input_buffer.ByteArr[0].7;

rfid_input_bitheader_2.CP := rfid_input_buffer.ByteArr[0].0;
rfid_input_bitheader_2.AA := rfid_input_buffer.ByteArr[0].1;
rfid_input_bitheader_2.AE := rfid_input_buffer.ByteArr[0].2;
rfid_input_bitheader_2.AF := rfid_input_buffer.ByteArr[0].3;
rfid_input_bitheader_2.Bit4 := rfid_input_buffer.ByteArr[0].4;
rfid_input_bitheader_2._TO := rfid_input_buffer.ByteArr[0].5;
rfid_input_bitheader_2.HF := rfid_input_buffer.ByteArr[0].6;
rfid_input_bitheader_2.BB := rfid_input_buffer.ByteArr[0].7;

rfid_output_buffer.ByteArr[0].0 := rfid_output_bitheader_1.AV ;
rfid_output_buffer.ByteArr[0].1 := rfid_output_bitheader_1.Bit1;
rfid_output_buffer.ByteArr[0].2 := rfid_output_bitheader_1.GR;
rfid_output_buffer.ByteArr[0].3 := rfid_output_bitheader_1.Bit3;
rfid_output_buffer.ByteArr[0].4 := rfid_output_bitheader_1.Bit4;
rfid_output_buffer.ByteArr[0].5 := rfid_output_bitheader_1.KA;
rfid_output_buffer.ByteArr[0].6 := rfid_output_bitheader_1.TI;
rfid_output_buffer.ByteArr[0].7 := rfid_output_bitheader_1.Bit7;

rfid_output_buffer.ByteArr[9].0 := rfid_output_bitheader_2.AV ;
rfid_output_buffer.ByteArr[9].1 := rfid_output_bitheader_2.Bit1;
rfid_output_buffer.ByteArr[9].2 := rfid_output_bitheader_2.GR;
rfid_output_buffer.ByteArr[9].3 := rfid_output_bitheader_2.Bit3;
rfid_output_buffer.ByteArr[9].4 := rfid_output_bitheader_2.Bit4;
rfid_output_buffer.ByteArr[9].5 := rfid_output_bitheader_2.KA;
rfid_output_buffer.ByteArr[9].6 := rfid_output_bitheader_2.TI;
rfid_output_buffer.ByteArr[9].7 := rfid_output_bitheader_2.Bit7;


IF rfid_start_toggle
THEN
	rfid_output_bitheader_1.GR := FALSE;
	rfid_output_bitheader_1.KA := FALSE;
	rfid_output_bitheader_1.AV := FALSE;
	rfid_output_bitheader_2.GR := FALSE;
	rfid_output_bitheader_2.KA := FALSE;
	rfid_output_bitheader_2.AV := FALSE;
	
	rfid_start_toggle := FALSE;
END_IF


IF 	rfid_shutdown_toggle
THEN
	rfid_output_bitheader_1.KA := TRUE;
	rfid_output_bitheader_2.KA := TRUE;
	
	IF 	rfid_input_bitheader_1.HF
		AND rfid_input_bitheader_2.HF
		AND NOT rfid_input_bitheader_1.CP
		AND NOT rfid_input_bitheader_2.CP
	THEN
		rfid_output_bitheader_1.KA := FALSE;
		rfid_output_bitheader_2.KA := FALSE;
		rfid_shutdown_toggle := FALSE;
	END_IF
		
END_IF


IF 	rfid_write_toggle //OR i_rfid_write_from_hmi
THEN	
	rfid_output_buffer.ByteArr[1] := 16#0032;
	rfid_output_buffer.ByteArr[2] := 16#00;
	rfid_output_buffer.ByteArr[3] := 16#00;
	rfid_output_buffer.ByteArr[4] := 16#0001;
	rfid_output_buffer.ByteArr[5] := 16#00;
	rfid_output_buffer.ByteArr[6] := rfid_value_to_write;
	
	rfid_output_bitheader_1.AV := TRUE;
	rfid_output_bitheader_2.AV := TRUE;
		
	IF 	rfid_input_bitheader_1.AA 
		AND rfid_input_bitheader_2.AA 
		AND rfid_input_bitheader_1.AE
		AND rfid_input_bitheader_2.AE
	THEN
		rfid_output_bitheader_1.AV := FALSE;
		rfid_output_bitheader_2.AV := FALSE;
		rfid_write_toggle := FALSE;
	END_IF
		
END_IF


IF 	rfid_read_toggle 
THEN	
	rfid_output_buffer.ByteArr[1] := 16#0001;
	rfid_output_buffer.ByteArr[2] := 16#00;
	rfid_output_buffer.ByteArr[3] := 16#00;
	rfid_output_buffer.ByteArr[4] := 16#0001;
	rfid_output_buffer.ByteArr[5] := 16#00;
	
	rfid_output_bitheader_1.AV := TRUE;
	rfid_output_bitheader_2.AV := TRUE;
	
	
	IF 	rfid_input_bitheader_1.AA 
		AND rfid_input_bitheader_2.AA 
		AND rfid_input_bitheader_1.AE
		AND rfid_input_bitheader_2.AE
	THEN
		// SAVE VALUES IN INPUT BUFFER [1...8] - CHECK WITH BRAND FOR WHAT VALUE SHOULD BE PRESENT
		rfid_value := rfid_input_buffer.ByteArr[1];
		rfid_output_bitheader_1.AV := FALSE;
		rfid_output_bitheader_2.AV := FALSE;
		rfid_read_toggle := FALSE;
	END_IF
	
END_IF



(* STATE MACHINE FOR READING AND WRITING TO RFID *)
CASE RFID_read_write_status OF
			
	CSP_CASE_LOADER_RFID_STATUS_START:
	
		IF csp_main_accuChange.RFID_read_write_running (* Use this value within brand change to start the check *)
		THEN
			rfid_write_done := FALSE;
			rfid_read_done := FALSE;
			rfid_read_write_running := TRUE;
			RFID_read_write_status_next := CSP_CASE_LOADER_RFID_STATUS_CHECK_AXIS_POS;
		END_IF
		
		
	CSP_CASE_LOADER_RFID_STATUS_CHECK_AXIS_POS:
	
		IF 	ABS(axis.actual_position - rfid_check_pos) < check_pls_tolerance
		THEN
			RFID_read_write_status_next := CSP_CASE_LOADER_RFID_STATUS_CHECK_READ_WRITE;
		ELSE
			RFID_read_write_status_next := CSP_CASE_LOADER_RFID_STATUS_DISABLE_AXIS;
		END_IF
		
	
	CSP_CASE_LOADER_RFID_STATUS_DISABLE_AXIS:
	
		axis_disable(axis);
		IF 	axis_is_disabled(axis)
		THEN
			RFID_read_write_status_next := CSP_CASE_LOADER_RFID_STATUS_ENABLE_AXIS;
		END_IF
		
		
	CSP_CASE_LOADER_RFID_STATUS_ENABLE_AXIS:
	
		IF servo_on_condition
		THEN
			axis_enable(axis);
		END_IF
		
		IF 	axis_is_enabled(axis)
		THEN
			RFID_read_write_status_next := CSP_CASE_LOADER_RFID_STATUS_ENABLE_CROSSPUSHERS;
		END_IF
		
	CSP_CASE_LOADER_RFID_STATUS_ENABLE_CROSSPUSHERS:
	
		axis_enable(csp_transfer_crosspusher_horizontal.axis);
		axis_enable(csp_transfer_crosspusher_follower.axis);
		IF 	axis_is_enabled(csp_transfer_crosspusher_horizontal.axis)
			AND
			axis_is_enabled(csp_transfer_crosspusher_follower.axis)
		THEN
			RFID_read_write_status_next := CSP_CASE_LOADER_RFID_STATUS_MOVE_CROSSPUSHERS;
		END_IF
	
	CSP_CASE_LOADER_RFID_STATUS_MOVE_CROSSPUSHERS:
	
		IF 	axis_is_standstill(csp_transfer_crosspusher_horizontal.axis)
			AND
			axis_is_standstill(csp_transfer_crosspusher_follower.axis)
		THEN
			axis_move_absolute(
				position 		:= csp_transfer_crosspusher_horizontal.load_position,
				velocity 		:= phase_velocity_degps,
				direction		:= AXIS_SHORTEST_WAY,
				acceleration 	:= MOTOR_MAX_ACCELLERATION_DEGPS2,
				deceleration 	:= MOTOR_MAX_DECELLERATION_DEGPS2, 
				jerk 			:= MOTOR_MAX_JERK_DEGPS3, 
				buffer_mode 	:= AXIS_BUFFER_MODE_BUFFERED,
				CONVERSION_this := csp_transfer_crosspusher_horizontal.axis
				); 
				
			axis_move_absolute(
				position 		:= 500,
				velocity 		:= phase_velocity_degps,
				direction		:= AXIS_SHORTEST_WAY,
				acceleration 	:= MOTOR_MAX_ACCELLERATION_DEGPS2,
				deceleration 	:= MOTOR_MAX_DECELLERATION_DEGPS2, 
				jerk 			:= MOTOR_MAX_JERK_DEGPS3, 
				buffer_mode 	:= AXIS_BUFFER_MODE_BUFFERED,
				CONVERSION_this := csp_transfer_crosspusher_follower.axis
				); 
		END_IF
			
		IF	axis_is_absolute_moving(csp_transfer_crosspusher_follower.axis) 
			OR
			axis_is_absolute_moving(csp_transfer_crosspusher_horizontal.axis) 
		THEN
			RFID_read_write_status_next := CSP_CASE_LOADER_RFID_VERIFY_CROSSPUSHERS_CLEAR;
		END_IF
	
		
	CSP_CASE_LOADER_RFID_VERIFY_CROSSPUSHERS_CLEAR:
	
		IF 	csp_transfer_crosspusher_horizontal.axis.actual_position >= csp_transfer_crosspusher_horizontal.load_position
			AND csp_transfer_crosspusher_follower.axis.actual_position >= (csp_transfer_crosspusher_follower.slave_scaling-1)
			OR
			(
				rfid_input_bitheader_1.CP 
				AND rfid_input_bitheader_2.CP
			)
		THEN
			RFID_read_write_status_next := CSP_CASE_LOADER_RFID_STATUS_MOVE_AXIS_TO_POS;
		END_IF
	
		
	CSP_CASE_LOADER_RFID_STATUS_MOVE_AXIS_TO_POS:

		
		IF 	axis_is_standstill(axis)
			AND
			axis_is_standstill(csp_transfer_crosspusher_horizontal.axis)
			AND
			axis_is_standstill(csp_transfer_crosspusher_follower.axis)
		THEN
			axis_move_absolute(
				position 		:= rfid_check_pos,
				velocity 		:= phase_velocity_degps,
				direction		:= AXIS_SHORTEST_WAY,
				acceleration 	:= MOTOR_MAX_ACCELLERATION_DEGPS2,
				deceleration 	:= MOTOR_MAX_DECELLERATION_DEGPS2, 
				jerk 			:= MOTOR_MAX_JERK_DEGPS3, 
				buffer_mode 	:= AXIS_BUFFER_MODE_BUFFERED,
				CONVERSION_this := axis
				); 
		END_IF
	
		IF 	axis_is_absolute_moving(axis) OR axis.actual_position <= rfid_check_pos
		THEN
			RFID_read_write_status_next := CSP_CASE_LOADER_RFID_STATUS_VERIFY_AXIS_POS;
		END_IF
		
		
	CSP_CASE_LOADER_RFID_STATUS_VERIFY_AXIS_POS:
	
		IF 	axis_is_standstill(axis)
			AND ABS(axis.actual_position - rfid_check_pos) < check_pls_tolerance
		THEN
			RFID_read_write_status_next := CSP_CASE_LOADER_RFID_STATUS_CHECK_READ_WRITE;
		END_IF
		
		
	(* CHECK IF IT IS SUPPOSED TO READ OR WRITE *)
	CSP_CASE_LOADER_RFID_STATUS_CHECK_READ_WRITE:
	
		rfid_start_toggle := TRUE;
		IF 	csp_main_accuChange.RFID_reading (* Use this value also within brand change *)
		THEN
			RFID_read_write_status_next := CSP_CASE_LOADER_RFID_STATUS_READ_START;
		ELSIF csp_main_accuChange.RFID_writing
		THEN
			RFID_read_write_status_next := CSP_CASE_LOADER_RFID_STATUS_WRITE_START;
		END_IF
			
		
		
	(* RFID READ START *)	
	CSP_CASE_LOADER_RFID_STATUS_READ_START:
	
		IF 	rfid_input_bitheader_1.CP
			AND rfid_input_bitheader_2.CP
		THEN
			rfid_read_toggle := TRUE;
			RFID_read_write_status_next := CSP_CASE_LOADER_RFID_STATUS_READ_CHECK_RESULT;
		END_IF

	CSP_CASE_LOADER_RFID_STATUS_READ_CHECK_RESULT:
	
		IF 	NOT rfid_read_toggle 
		THEN
			RFID_read_write_status_next := CSP_CASE_LOADER_RFID_STATUS_READ_DONE;
		END_IF
		
	CSP_CASE_LOADER_RFID_STATUS_READ_DONE:
	
		rfid_read_done := TRUE;
		rfid_read_write_running := FALSE;
		RFID_read_write_status_next := CSP_CASE_LOADER_RFID_STATUS_WAITING;
		
		
	(* RFID WRITING START *)
	CSP_CASE_LOADER_RFID_STATUS_WRITE_START:
	
		rfid_value_to_write := csp_main_accuChange.RFID_Setup_write_value;
		
		IF	rfid_input_bitheader_1.CP
			AND rfid_input_bitheader_2.CP
		THEN
			rfid_write_toggle := TRUE;
			RFID_read_write_status_next := CSP_CASE_LOADER_RFID_STATUS_WAIT_WRITE;
		END_IF
		
		
	CSP_CASE_LOADER_RFID_STATUS_WAIT_WRITE:
	
		IF 	NOT rfid_write_toggle
		THEN	
				RFID_read_write_status_next := CSP_CASE_LOADER_RFID_STATUS_WRITE_DONE;
		END_IF
		
	CSP_CASE_LOADER_RFID_STATUS_WRITE_DONE:
	
		rfid_write_done := TRUE;
		rfid_read_write_running := FALSE;
		RFID_read_write_status_next := CSP_CASE_LOADER_RFID_STATUS_WAITING;
		
		
	CSP_CASE_LOADER_RFID_STATUS_WAITING:
	
		RFID_read_write_status_next := CSP_CASE_LOADER_RFID_STATUS_START;
		
	
END_CASE


(* ADVANCES TO NEXT STEP *)
IF 	NOT RFID_read_write_debug
	OR
	RFID_read_write_one_step	
THEN
	RFID_read_write_status := RFID_read_write_status_next;
	RFID_read_write_one_step := FALSE;
END_IF


(* Connection timeout *)
IF	RFID_read_write_running
	AND NOT RFID_read_write_debug
THEN
	IF	timer_is_expired(RFID_read_write_tmr)
	THEN
		rfid_start_toggle := TRUE;
		process_message_set(1, RFID_read_write_status, 0, RFID_read_write_error_msg);
	END_IF
ELSE
	timer_restart(10000, RFID_read_write_tmr);
END_IF
END_ACTION

END_PROGRAM

// ---- Application/CSP/Main/AccU Change/csp_main_accuChange.TcPOU
(*********************************** G.D S.p.A. - Technical Department ***********************************
============= PROGRAM INFO ============
FOLDER:             TBD
MACHINES INVOLVED:  TBD 

============= DESCRIPTION =============
csp brand management program

============= REVISIONS ===============
Date		Version	 	Author      	Description             
----------	-------		------------  	--------------------------------------------
2020/02/12 	0000.00	 	G.Imbriaco		Common AccU Change enable/disable and velocity parameter
2020/05/07	0001.00		M.Peppo			Initial AccU Change Sequence Added

**********************************************************************************************************)
(*$R
	process_ref := prc;
$*)
PROGRAM csp_main_accuChange
VAR
	request_test:												BOOL;	
	test_in_position:											BOOL;
	
	first_scan_rtrig:											R_Trig;
	first_scan_bool:											BOOL := FALSE;
	
	not_in_brand_change:										BOOL;  (*$P $*)
	brand_change_check_string:									STRING := ''; (*$P $*)
	brand_change_check_delay_tmr:								timer;
	
	machine_ready_and_enable:                                   BOOL := FALSE; 
	hmi_machine_ready_and_enable_hgos:							hmi_graphic_object_status;
	
	prc:														process;
	prc_path:													STRING;	
	all_in_position_motcond:									motorization_conditioner;
	
	eoat_rfid_checked_motcond:									motorization_conditioner;
	loader_pusher_rfid_checked_motcond:							motorization_conditioner;
	loader_plate_rfid_checked_motcond:							motorization_conditioner;
	
	cam_data_changed:											BOOL;
	
	null_byte:													BYTE;
	size_change_in_middle_of_changeover:						BOOL := FALSE;
	
	manual_empty:												BOOL;
	manual_empty_cbtn:											command_button;

	brand_change_request_dvr:									BOOL;
	brand_change_request_cbtn:									command_button;

	running_rfid_status:										csp_main_accuChange_RFID_running_check_status;
	running_rfid_status_next:									csp_main_accuChange_RFID_running_check_status;
	
	
	fsm_status:													csp_main_accuChange_enum;(*$M $*)
	fsm_next_status:											csp_main_accuChange_enum;
	fsm_enable_condition:										BOOL:=FALSE;
	
	fsm_conditions:												BOOL;
	fsm_running:												BOOL;
	fsm_timeout:												BOOL;

	fsm_tmr:													timer;
	
	debug_fsm:													BOOL := FALSE;
	debug_fsm_one_step:											BOOL := FALSE;
	
	changeover_timeout_asm:										message;
	navigate_custom_screen_aem:									message;
	change_parts_incorrect_aem:									message;
	
	buzzer_req_bool:											boolean;
	buzzer_req_tmr:												timer;
	stabilization_tmr:											timer;
	buzzer_test_bool:											BOOL;
	
	completed_bool:												boolean;
	change_bor:													boolean_or;
	
	start_btn:													BOOL;
	stop_btn:													BOOL;

	start_changeover:											BOOL; //Used for Step 3 onward
	
	p_brand_changeover_mode_enable:								BOOL;	(*$P $*)

	machine_size_running:										BOOL := FALSE;
	machine_empty:												BOOL := FALSE;
	
	Brand_Change_Occurred:										BOOL := FALSE;
	Case_Motors_Safe_accU:										BOOL := FALSE;
	
	RFID_check_request:											BOOL := FALSE;
	changeover_rfid_read_done:									BOOL := FALSE;
	changeover_rfid_write_done:									BOOL := FALSE;
	changeover_rfid_value:										BYTE;
	changover_rfid_read_write_running:							BOOL := FALSE;
	
	failed_change_part_verify_fault:							BOOL := FALSE; // ADD TO CSP LOGIC
	change_part_eoat_confirmed:									BOOL := FALSE; //REPLACE WITH CSP BIT
	change_part_pusher_confirmed:								BOOL := FALSE;
	change_part_plate_confirmed:								BOOL := FALSE;
	change_part_paddles_OS_confirmed:							BOOL := FALSE;
	change_part_paddles_LS_confirmed:							BOOL := FALSE;
	
	change_part_eoat_wrong:										message;
	change_part_pusher_wrong:									message;
	change_part_plate_wrong:									message;
	change_part_paddles_wrong:									message;
	
	Group_1_motors_request:										BOOL := FALSE; //If true all group 1 motors move to target position of new size
	Group_1_motors_in_position:									BOOL := FALSE;
	Group_2_motors_request:										BOOL := FALSE;	
	Group_2_motors_in_position:									BOOL := FALSE;
	
	(* ALL MOVE REQS *)
	case_transport_accU_depth_move_req:							BOOL := FALSE; // DONE
	
	case_feed_magazine_accU_lsDepth_move_req:					BOOL := FALSE; // DONE
	case_feed_magazine_accU_osDepth_move_req:					BOOL := FALSE; // DONE

	transfer_infeed_accU_depth_move_req:						BOOL := FALSE;
	transfer_infeed_accU_waterfall_move_req:					BOOL := FALSE; // DONE
	transfer_accumulator_accU_depth_move_req:					BOOL := FALSE; // DONE

	case_tr_accU_depth_move_req:								BOOL := FALSE;
	
	case_loader_guide_accU_width_move_req:						BOOL := FALSE; // DONE
	case_glue_os_accU_width_move_req:							BOOL := FALSE;
	case_glue_os_accU_upperPosition_move_req:					BOOL := FALSE;
	case_glue_os_accU_lowerPosition_move_req:					BOOL := FALSE;
	case_glue_ls_accU_upperPosition_move_req:					BOOL := FALSE;
	case_glue_ls_accU_lowerPosition_move_req:					BOOL := FALSE;
	
	case_tr_accU_ls_width_move_req:								BOOL := FALSE; // DONE
	
	
	
	
	motors_in_safe_pos_boolean:									boolean;
	stop_machine_for_change_parts_dchk:							digital_check;
	
	Motion_Motors_New_Size_Req:									BOOL := FALSE;//Pneumatic move request is part of this bit
	Case_Motors_In_New_Accu_Pos:								BOOL := FALSE;
	Motion_motors_in_position:									BOOL := FALSE;
	
	all_motors_in_position:										BOOL := FALSE;
	
	navigate_to_accU_popup:										BOOL := FALSE;
	navigate_to_accU_popup_dvr:									BOOL;
	navigate_to_accu_popup_cbtn:								command_button;
	
	
	remove_product_popup:										BOOL := FALSE;
	trigger_change_parts_incorrect_popup:						BOOL := FALSE;

	brand1_active:												BOOL := FALSE;
	brand2_active:												BOOL := FALSE;
	brand3_active:												BOOL := FALSE;
	brand4_active:												BOOL := FALSE;
	brand5_active:												BOOL := FALSE;
	brand6_active:												BOOL := FALSE;
	brand7_active:												BOOL := FALSE;
	brand8_active:												BOOL := FALSE;
	brand9_active:												BOOL := FALSE;
	brand10_active:												BOOL := FALSE;
	brand11_active:												BOOL := FALSE;
	brand12_active:												BOOL := FALSE;
	brand13_active:												BOOL := FALSE;
	brand14_active:												BOOL := FALSE;
	brand15_active:												BOOL := FALSE;
	brand16_active:												BOOL := FALSE;
	brand17_active:												BOOL := FALSE;
	brand18_active:												BOOL := FALSE;
	brand19_active:												BOOL := FALSE;	

	// HMI custom page variable management
	hmi_toggle_cbtn:											command_button;
	enable_write:												BOOL;
	hmi_toggle_counter:											INT := 0;
	hmi_brand_color_red:										BOOL := FALSE;
	hmi_brand_color_green:										BOOL := TRUE;
	hmi_toggle_bit:												BOOL := FALSE;
	hmi_toggle_hgos:											hmi_graphic_object_status;
	
	hmi_current_accU_step:										INT  := 0;
	hmi_accU_step1_on:											BOOL := FALSE;
	hmi_accU_step2_on:											BOOL := FALSE;
	hmi_accU_step3_on:											BOOL := FALSE;
	hmi_accU_step4_on:											BOOL := FALSE;
	hmi_accU_step5_on:											BOOL := FALSE;
	hmi_accU_step6_on:											BOOL := FALSE;
	hmi_accU_step7_on:											BOOL := FALSE;
	
	hmi_brand_status_color_hgos:								hmi_graphic_object_status;
	hmi_brand_status_bad_color_hgos:							hmi_graphic_object_status;
	hmi_accU_step1_on_hgos:										hmi_graphic_object_status;
	hmi_accU_step1_off_hgos:									hmi_graphic_object_status;
	hmi_accU_step2_on_hgos:										hmi_graphic_object_status;
	hmi_accU_step2_off_hgos:									hmi_graphic_object_status;
	hmi_accU_step3_on_hgos:										hmi_graphic_object_status;
	hmi_accU_step3_off_hgos:									hmi_graphic_object_status;
	hmi_accU_step4_on_hgos:										hmi_graphic_object_status;
	hmi_accU_step4_off_hgos:									hmi_graphic_object_status;
	hmi_accU_step5_on_hgos:										hmi_graphic_object_status;
	hmi_accU_step5_off_hgos:									hmi_graphic_object_status;
	hmi_accU_step6_on_hgos:										hmi_graphic_object_status;
	hmi_accU_step6_off_hgos:									hmi_graphic_object_status;
	hmi_accU_step7_on_hgos:										hmi_graphic_object_status;
	hmi_accU_step7_off_hgos:									hmi_graphic_object_status;
	
	hmi_in_position_on_hgos:									hmi_graphic_object_status;
	hmi_in_position_off_hgos:									hmi_graphic_object_status;

	//Motor setup screen indicators
    hmi_in_position_transport_depth_on_hgos:					hmi_graphic_object_status;
	hmi_in_position_transport_depth_off_hgos:					hmi_graphic_object_status;	
	hmi_in_position_shuttle_depth_on_hgos:					    hmi_graphic_object_status;
	hmi_in_position_shuttle_depth_off_hgos:					    hmi_graphic_object_status;	
	hmi_in_position_magazine_ls_depth_on_hgos:					hmi_graphic_object_status;
	hmi_in_position_magazine_ls_depth_off_hgos:					hmi_graphic_object_status;	
	hmi_in_position_magazine_os_depth_on_hgos:					hmi_graphic_object_status;
	hmi_in_position_magazine_os_depth_off_hgos:					hmi_graphic_object_status;	
	hmi_in_position_loader_guide_width_on_hgos:					hmi_graphic_object_status;
	hmi_in_position_loader_guide_width_off_hgos:				hmi_graphic_object_status;	
	hmi_in_position_glue_os_upper_on_hgos:						hmi_graphic_object_status;
	hmi_in_position_glue_os_upper_off_hgos:						hmi_graphic_object_status;	
	hmi_in_position_glue_os_lower_on_hgos:						hmi_graphic_object_status;
	hmi_in_position_glue_os_lower_off_hgos:						hmi_graphic_object_status;	
	hmi_in_position_glue_ls_upper_on_hgos:						hmi_graphic_object_status;
	hmi_in_position_glue_ls_upper_off_hgos:						hmi_graphic_object_status;	
	hmi_in_position_glue_ls_lower_on_hgos:						hmi_graphic_object_status;
	hmi_in_position_glue_ls_lower_off_hgos:						hmi_graphic_object_status;	
	hmi_in_position_glue_os_width_on_hgos:						hmi_graphic_object_status;
	hmi_in_position_glue_os_width_off_hgos:						hmi_graphic_object_status;	
	hmi_in_position_transfer_infeed_depth_on_hgos:				hmi_graphic_object_status;
	hmi_in_position_transfer_infeed_depth_off_hgos:				hmi_graphic_object_status;	
	hmi_in_position_waterfall_on_hgos:							hmi_graphic_object_status;
	hmi_in_position_waterfall_off_hgos:							hmi_graphic_object_status;	
	hmi_in_position_accumulator_depth_on_hgos:					hmi_graphic_object_status;
	hmi_in_position_accumulator_depth_off_hgos:					hmi_graphic_object_status;	
	hmi_in_position_accumulator_conv_depth_on_hgos:				hmi_graphic_object_status;
	hmi_in_position_accumulator_conv_depth_off_hgos:				hmi_graphic_object_status;	
	hmi_in_position_top_rail_os_width_on_hgos:					hmi_graphic_object_status;
	hmi_in_position_top_rail_os_width_off_hgos:					hmi_graphic_object_status;	
	hmi_in_position_top_rail_ls_width_on_hgos:					hmi_graphic_object_status;
	hmi_in_position_top_rail_ls_width_off_hgos:					hmi_graphic_object_status;	
	hmi_in_position_top_rail_depth_on_hgos:						hmi_graphic_object_status;
	hmi_in_position_top_rail_depth_off_hgos:					hmi_graphic_object_status;	
	hmi_in_position_discharge_os_depth_on_hgos:					hmi_graphic_object_status;
	hmi_in_position_discharge_os_depth_off_hgos:				hmi_graphic_object_status;	
	
	
	
	//Case Feed EOAT Change Part
	change_part_color:											csp_main_accuChange_partColor_enum;
	hmi_change_part_eoat_color:									csp_main_accuChange_partColor_enum;
	hmi_change_part_eoat_red_on:								BOOL := FALSE;
	hmi_change_part_eoat_green_on:								BOOL := FALSE;
	hmi_change_part_eoat_blue_on:								BOOL := FALSE;
	hmi_change_part_eoat_yellow_on:								BOOL := FALSE;
	hmi_change_part_eoat_white_on:								BOOL := FALSE;
	hmi_change_part_eoat_black_on:								BOOL := FALSE;
	hmi_change_part_eoat_orange_on:								BOOL := FALSE;
	hmi_change_part_eoat_checkbox_on:							BOOL := FALSE;
	hmi_change_part_eoat_red_hgos:								hmi_graphic_object_status;
	hmi_change_part_eoat_green_hgos:							hmi_graphic_object_status;
	hmi_change_part_eoat_blue_hgos:								hmi_graphic_object_status;
	hmi_change_part_eoat_yellow_hgos:							hmi_graphic_object_status;
	hmi_change_part_eoat_white_hgos:							hmi_graphic_object_status;
	hmi_change_part_eoat_black_hgos:							hmi_graphic_object_status;
	hmi_change_part_eoat_orange_hgos:							hmi_graphic_object_status;
	hmi_change_part_eoat_checkbox_hgos:							hmi_graphic_object_status;
	//Loader Pusher Change Part
	hmi_change_part_pusher_color:								csp_main_accuChange_partColor_enum;
	hmi_change_part_pusher_green_on:							BOOL := FALSE;
	hmi_change_part_pusher_yellow_on:							BOOL := FALSE;
	hmi_change_part_pusher_white_on:							BOOL := FALSE;
	hmi_change_part_pusher_black_on:							BOOL := FALSE;
	hmi_change_part_pusher_checkbox_on:							BOOL := FALSE;
	hmi_change_part_pusher_green_hgos:							hmi_graphic_object_status;
	hmi_change_part_pusher_yellow_hgos:							hmi_graphic_object_status;
	hmi_change_part_pusher_white_hgos:							hmi_graphic_object_status;
	hmi_change_part_pusher_black_hgos:							hmi_graphic_object_status;
	hmi_change_part_pusher_checkbox_hgos:						hmi_graphic_object_status;
	//Loader Guide Plate Change Part
	hmi_change_part_plate_color:								csp_main_accuChange_partColor_enum;
	hmi_change_part_plate_green_on:								BOOL := FALSE;
	hmi_change_part_plate_yellow_on:							BOOL := FALSE;
	hmi_change_part_plate_black_on:								BOOL := FALSE;
	hmi_change_part_plate_checkbox_on:							BOOL := FALSE;
	hmi_change_part_plate_green_hgos:							hmi_graphic_object_status;
	hmi_change_part_plate_yellow_hgos:							hmi_graphic_object_status;
	hmi_change_part_plate_black_hgos:							hmi_graphic_object_status;
	hmi_change_part_plate_checkbox_hgos:						hmi_graphic_object_status;
	
	//Closing Paddle Change Part
	//No Current Color Blocks - Reserved for future
	hmi_change_part_paddle_color:								csp_main_accuChange_partColor_enum;
	hmi_change_part_paddle_checkbox_on:							BOOL := FALSE;
	hmi_change_part_paddle_checkbox_hgos:						hmi_graphic_object_status;
	
	RFID_Setup_write_value:										BYTE;
	RFID_Setup_read_value:										BYTE;
	RFID_Setup_read_value_string:								STRING;		(*$M desc := Read value to display on HMI; $*)
	RFID_Setup_read_cbtn:										command_button;
	RFID_Setup_write_cbtn:										command_button;
	
	RFID_reader_list_accuchange:								csp_main_accUChange_RFID_reader_list;	(*$P desc := Acc-U-Change RFID Reader selection list; $*)
	RFID_reader_list_accuchange_old:							csp_main_accUChange_RFID_reader_list;
	RFID_reader_brand_colors:									csp_main_accuChange_partColor_enum; 	(*$P desc := Acc-U-Change RFID Color selection list; $*)
	
	RFID_reading:												BOOL;
	RFID_writing:												BOOL;
	
	RFID_read_write_status:										csp_main_accuChange_RFID_read_write_status;
	RFID_read_write_status_next:								csp_main_accuChange_RFID_read_write_status;
	RFID_read_write_debug:										BOOL := FALSE;
	RFID_read_write_one_step:									BOOL := FALSE;
	RFID_read_write_running:									BOOL;
	RFID_read_write_tmr:										timer;
	RFID_read_write_error_msg:									message;
	
	//Bold Text to highlight current step
	//hmi_step1_bold_hgos
	closing_horizontal_safe: 									BOOL := FALSE;						
	loader_in_position: 										BOOL;
	case_feed_in_position: 										BOOL;
	closing_os_in_position: 									BOOL;
	closing_ls_in_position: 									BOOL;
	loader_plate_in_position: 									BOOL;
	change_part_in_position: 									BOOL;
		
	accU_axis_moving:											BOOL;
	accU_axis_moving_horn_on:									BOOL;
	horn_on_filter:												filter;
	
	horn_on_time:												DINT := 3000; (*$P $*)
	horn_off_time:												DINT := 100; (*$P $*)
	
	bypass_paddle: 												BOOL := True;
	Initial_Commissioning_bit: 									BOOL := False;
END_VAR

VAR CONSTANT
	CONSTANTS:													csp_main_accuChange_constant;
	CHANGEOVER_TIMEOUT_S:										INT := 360;
	BUZZER_REQ_TIMEOUT_S:										INT := 3;
	STABILIZATION_TIMEOUT_S:									INT := 3;
END_VAR

VAR PERSISTENT
	machine_size_complete:										BOOL := true;
END_VAR

_read_var_input();

_object_manager();

IF NOT objects_running()
THEN
	RETURN;	
END_IF

_read_process_image();

_mode_manager();

CASE process_get_mode(prc) OF
	MODE_ABSENT,
	MODE_INACTIVE:
		RETURN;
	MODE_TEST:
		_handle_process_test();
END_CASE

//first_scan_rtrig(CLK := power_done);

_set_runtime_properties();
_brand_colors();
_in_position();
_hmi_management();
RFID();

(********************************* BODY *********************************)

(* VERIFIES ALL ACC-U-CHANGE MOTORS ARE IN POSITION BEFORE EVERY RUN *)
IF 	machine_size_complete
	AND
	(
	Group_1_motors_in_position
	AND Group_2_motors_in_position
	OR Initial_Commissioning_bit
	)
THEN
	motorization_conditioner_start_done(all_in_position_motcond);
END_IF


(* USED TO CHANGE VISIBILITY ON MESSAGE FOR RFID *)
IF machine_is_ready(csp.mch)
	OR
	(RFID_reader_list_accuchange = CASE_FEED_EOAT_READER
	AND
	csp_case_feed_arm_sensors.rfid_input_bitheader_1.CP
	AND
	csp_case_feed_arm_sensors.rfid_input_bitheader_2.CP)
	OR
	(RFID_reader_list_accuchange = LOADER_PUSHER_READER
	AND
	csp_case_loader_pusher.rfid_input_bitheader_1.CP
	AND
	csp_case_loader_pusher.rfid_input_bitheader_2.CP)
	OR
	(RFID_reader_list_accuchange = LOADER_GUIDE_PLATE_READER
	AND
	csp_case_loader_sensors.rfid_input_bitheader_1.CP
	AND
	csp_case_loader_sensors.rfid_input_bitheader_2.CP)
THEN
	machine_ready_and_enable := TRUE;
ELSE
	machine_ready_and_enable := FALSE;               
END_IF

	hmi_graphic_object_set_status(
        status  			:= SEL(machine_ready_and_enable, HMI_OBJECT_STATUS_INVISIBLE, HMI_OBJECT_STATUS_ON),
        CONVERSION_this     := hmi_machine_ready_and_enable_hgos);

(*  *)
IF Brand_Change_Occurred
THEN
	RFID_read_write_status := READ_WRITE_STATUS_ERROR;
END_IF


(* BUTTON ACTIVATION TO MOVE MACHINE TO CLEANOUT MODE *)
IF command_button_get_actual_value(manual_empty_cbtn) = HMI_BUTTON_STATUS_ON
THEN
	manual_empty := TRUE;
ELSE
	manual_empty := FALSE;
END_IF


(* CHECKS IF A BRAND CHANGE IS INITIATED IN THE MIDDLE OF A SIZE CHANGE AND RESETS *)
IF 	csp_main_brand.count_changed
	AND NOT machine_size_complete
THEN
	fsm_next_status := CSP_MAIN_ACCUCHANGE_STATUS_BRAND_CHECK;
	size_change_in_middle_of_changeover := TRUE;
END_IF

(* CLEARS ERROR RFID HANDLING *)
IF machine_get_reset_edge(csp.mch)
THEN
	process_message_reset(change_part_eoat_wrong);
	process_message_reset(change_part_pusher_wrong);
	process_message_reset(change_part_plate_wrong);
	process_message_reset(change_part_paddles_wrong);
END_IF

(* RUNS AT THE BEGINNING OF aHMI STARTUP WAITING FOR PARAMETER TO LAOD SO THAT SIZE CHANGE DOESN'T OVERWRITE WHEN NO CHANGE *)
//brand_change_check_string := csp_main_brand.count;
IF brand_change_check_string = ''
THEN
	timer_restart(5000, brand_change_check_delay_tmr);
END_IF



IF 	not_in_brand_change
	OR first_scan_rtrig.q
THEN
	machine_size_complete := TRUE;
	hmi_current_accU_step := 0;
	Brand_Change_Occurred := FALSE;
	navigate_to_accU_popup := FALSE;
	cam_data_changed := FALSE;
	fsm_next_status := CSP_MAIN_ACCUCHANGE_STATUS_BRAND_CHECK;
	
	not_in_brand_change := FALSE;
END_IF


fsm_enable_condition := 
						process_is_ready(prc)
						AND 
						(*process_subtree_is_ready(prc)
						AND*)
						process_get_mode(csp_main_accuChange.prc) = MODE_OPERATIONAL
						AND
						csp_main_brand.count <> ''; //Brand_Change_Occurred; //csp_main_brand.count_changed;
					
IF NOT fsm_enable_condition
THEN
	fsm_status	:=	CSP_MAIN_ACCUCHANGE_STATUS_BRAND_CHECK;
END_IF


CASE fsm_status OF
	CSP_MAIN_ACCUCHANGE_STATUS_BRAND_CHECK:
		
		IF	(
				machine_download_is_running(csp.mch)
				OR 
				size_change_in_middle_of_changeover
			)
			AND first_scan_bool
		THEN
			navigate_to_accU_popup := TRUE;
			fsm_next_status := CSP_MAIN_ACCUCHANGE_STATUS_BRAND_CHANGE_REQUEST;
		END_IF
		
		
	CSP_MAIN_ACCUCHANGE_STATUS_BRAND_CHANGE_REQUEST:
	
		IF brand_change_request_dvr
		THEN
			hmi_current_accU_step := 1;
			machine_size_complete := FALSE;
			Motion_Motors_New_Size_Req := FALSE;
			Brand_Change_Occurred := TRUE;
			size_change_in_middle_of_changeover := FALSE;
			
			change_part_eoat_confirmed := FALSE;
			change_part_pusher_confirmed := FALSE;
			change_part_plate_confirmed := FALSE;
			change_part_paddles_OS_confirmed := FALSE;
			change_part_paddles_LS_confirmed := FALSE;
			
			hmi_change_part_eoat_checkbox_on := FALSE;
			hmi_change_part_pusher_checkbox_on := FALSE;
			hmi_change_part_plate_checkbox_on := FALSE;
			hmi_change_part_paddle_checkbox_on := FALSE;
			
			fsm_next_status := CSP_MAIN_ACCUCHANGE_STATUS_PRODUCT_REMOVED_CHECK;
		END_IF
		
		
	CSP_MAIN_ACCUCHANGE_STATUS_PRODUCT_REMOVED_CHECK:
	
		IF 	machine_empty
			AND machine_is_stop_emergency_active(csp.mch)
		THEN
			cam_data_changed := TRUE;
			fsm_next_status := CSP_MAIN_ACCUCHANGE_STATUS_RESET_REQUEST;
		ELSE
			remove_product_popup := TRUE; //"Please remove product" to Operator //Currently not being called ... Should this be a fault instead? CALL THIS MANUAL EMPTY AND PUT ON ACCU SCREEN
		END_IF
		
		
	CSP_MAIN_ACCUCHANGE_STATUS_RESET_REQUEST:
	
		IF machine_is_stopped(csp.mch)
		THEN
			hmi_current_accU_step := 2; //"RESET AND START Machine"
			fsm_next_status := CSP_MAIN_ACCUCHANGE_STATUS_SAFE_POSITION_REQUEST;
		END_IF
		
		
	CSP_MAIN_ACCUCHANGE_STATUS_SAFE_POSITION_REQUEST:
	
		IF machine_is_running(csp.mch)
		THEN
			hmi_current_accU_step:= 3; //"Machine Moves to Change Part Removal Position"
			fsm_next_status := CSP_MAIN_ACCUCHANGE_STATUS_OPERATOR_REPLACE_CHANGE_PARTS;
		END_IF
		
		
	CSP_MAIN_ACCUCHANGE_STATUS_OPERATOR_REPLACE_CHANGE_PARTS: 
	
		IF 	Case_Motors_Safe_accU
			AND machine_is_running(csp.mch)
		THEN
			boolean_set(motors_in_safe_pos_boolean);
			hmi_current_accU_step:= 4; //"Replace Specified Change Parts AND RESET AND START"
			fsm_next_status := CSP_MAIN_ACCUCHANGE_STATUS_CHANGE_PARTS_REPLACED;
		END_IF
		
		
	CSP_MAIN_ACCUCHANGE_STATUS_CHANGE_PARTS_REPLACED:
		
		boolean_reset(motors_in_safe_pos_boolean);
		
		IF machine_is_ready(csp.mch)
		THEN
			// ADD MESSAGE TO TELL THEM TO RESET AND START MACHINE
			fsm_next_status := CSP_MAIN_ACCUCHANGE_STATUS_VERIFYING_CHANGE_PARTS_START;
		END_IF
		
		
	CSP_MAIN_ACCUCHANGE_STATUS_VERIFYING_CHANGE_PARTS_START:
	
		hmi_current_accU_step:= 5; //"Verifying Change Parts"
		RFID_check_request := TRUE;
		
		(* ENABLES CHECK REQUEST FOR RFID IN A STEP BY STEP ORDER STARTING WITH CASE_FEED_EOAT_READER *)
		IF RFID_check_request
		THEN
			RFID_reader_list_accuchange := NO_READER_SELECTED;
			RFID_read_write_running := TRUE;
			RFID_reading := TRUE;
			
			fsm_next_status := CSP_MAIN_ACCUCHANGE_STATUS_VERIFYING_CASE_FEED_EOAT;			
		END_IF
		
		
	CSP_MAIN_ACCUCHANGE_STATUS_VERIFYING_CASE_FEED_EOAT:
	
		RFID_reader_list_accuchange := CASE_FEED_EOAT_READER;
		
		(* PRODUCTION LOGIC *)
		IF 	NOT change_part_eoat_confirmed
			AND NOT process_message_is_on(change_part_eoat_wrong)
		THEN
			RFID_reading := TRUE;
		END_IF
		
		
		IF csp_case_feed_arm_sensors.rfid_read_done
		THEN
			RFID_reading := FALSE;
			
			IF changeover_rfid_value = INT_TO_BYTE(hmi_change_part_eoat_color)
			THEN
				change_part_eoat_confirmed := TRUE;
				hmi_change_part_eoat_checkbox_on := TRUE;
				fsm_next_status := CSP_MAIN_ACCUCHANGE_STATUS_VERIFYING_LOADER_PUSHER; (* MOVES TO LOADER_GUIDE_PUSHER_READER *)
			ELSE
				process_message_set(1, 0, 0, change_part_eoat_wrong);
			END_IF
		END_IF
			
		
	CSP_MAIN_ACCUCHANGE_STATUS_VERIFYING_LOADER_PUSHER:
	
		RFID_reader_list_accuchange := LOADER_PUSHER_READER;
		
		IF NOT change_part_pusher_confirmed
			AND NOT process_message_is_on(change_part_pusher_wrong)
		THEN
			RFID_reading := TRUE;
		END_IF
				
		IF csp_case_loader_pusher.rfid_read_done
		THEN
			RFID_reading := FALSE;
			
			IF changeover_rfid_value = INT_TO_BYTE(hmi_change_part_pusher_color)
			THEN
				change_part_pusher_confirmed := TRUE;
				hmi_change_part_pusher_checkbox_on := TRUE;
				fsm_next_status := CSP_MAIN_ACCUCHANGE_STATUS_VERIFYING_LOADER_GUIDE_PLATE; (* MOVES TO LOADER_GUIDE_PLATE_READER *)
			ELSE
				process_message_set(1, 0, 0, change_part_pusher_wrong);
			END_IF
		END_IF
		
		
	CSP_MAIN_ACCUCHANGE_STATUS_VERIFYING_LOADER_GUIDE_PLATE:
	
		RFID_reader_list_accuchange := LOADER_GUIDE_PLATE_READER;
		
		IF 	NOT change_part_plate_confirmed
			AND NOT process_message_is_on(change_part_plate_wrong)
		THEN
			RFID_reading := TRUE;
		END_IF
		
		IF csp_case_loader_sensors.rfid_read_done
		THEN
			RFID_reading := FALSE;
			
			IF changeover_rfid_value = INT_TO_BYTE(hmi_change_part_plate_color)
			THEN
				change_part_plate_confirmed := TRUE;
				hmi_change_part_plate_checkbox_on := TRUE;
				fsm_next_status := CSP_MAIN_ACCUCHANGE_STATUS_VERIFYING_CLOSING_PADDLES; (* MOVES TO CLOSING PADDLES READER *)
			ELSE
				process_message_set(1, 0, 0, change_part_plate_wrong);
			END_IF
		END_IF
			
				
	CSP_MAIN_ACCUCHANGE_STATUS_VERIFYING_CLOSING_PADDLES:
	
		RFID_reader_list_accuchange := CLOSING_PADDLES_READER;
		
		IF	NOT change_part_paddles_OS_confirmed
			AND NOT change_part_paddles_LS_confirmed
			AND NOT process_message_is_on(change_part_pusher_wrong)
		THEN
			RFID_reading := TRUE;
		END_IF
		
		IF csp_case_closing.rfid_read_done
			 //manual bypass added 05/10/21
			THEN
				RFID_reading := FALSE;
				
				IF changeover_rfid_value = INT_TO_BYTE(hmi_change_part_paddle_color)
				THEN
					change_part_paddles_OS_confirmed := TRUE;
					change_part_paddles_LS_confirmed := TRUE;
					
					hmi_change_part_paddle_checkbox_on := TRUE;
					fsm_next_status := CSP_MAIN_ACCUCHANGE_STATUS_VERIFYING_ALL_RFID;
				ELSE
					process_message_set(1, 0, 0, change_part_paddles_wrong);
				END_IF
		END_IF
		//Remove logic when paddle RFID can be reached by servo motors
		IF bypass_paddle
		THEN
			change_part_paddles_OS_confirmed := TRUE;
			change_part_paddles_LS_confirmed := TRUE;
			hmi_change_part_paddle_checkbox_on := TRUE;
			fsm_next_status := CSP_MAIN_ACCUCHANGE_STATUS_VERIFYING_ALL_RFID;
		END_IF
			
		
	CSP_MAIN_ACCUCHANGE_STATUS_VERIFYING_ALL_RFID:
	
		RFID_read_write_running := FALSE;
		RFID_reading := FALSE;
		
		IF 	change_part_eoat_confirmed
			AND change_part_pusher_confirmed
			AND change_part_plate_confirmed
			AND change_part_paddles_OS_confirmed
			AND change_part_paddles_LS_confirmed
		THEN
			cam_data_changed := FALSE;
			hmi_current_accU_step:= 6; //"Machine Moves to Selected Brand"
			fsm_next_status := CSP_MAIN_ACCUCHANGE_STATUS_GROUP_1_ACCU_MOVE_REQUEST;
		END_IF
		
		
	CSP_MAIN_ACCUCHANGE_STATUS_GROUP_1_ACCU_MOVE_REQUEST:
				
		(* ACCUMULATOR VM MOVE *)
		IF 	NOT csp_transfer_accumulator_accU_depth.in_position
			AND NOT csp_transfer_accumulator_accU_convDepth.in_position
		THEN
			transfer_accumulator_accU_depth_move_req := TRUE;
		END_IF
		
		IF 	csp_transfer_accumulator_accU_depth.in_position
			AND csp_transfer_accumulator_accU_convDepth.in_position
		THEN
			transfer_accumulator_accU_depth_move_req := FALSE;
		END_IF
		
		(* INFEED GUIDE DEPTH MOVE *)
		IF NOT csp_transfer_infeed_accU_depth.in_position
		THEN
			transfer_infeed_accU_depth_move_req := TRUE;
		ELSE
			IF axis_is_disabled(csp_transfer_infeed_accU_depth.axis)
			THEN
				transfer_infeed_accU_depth_move_req := FALSE;
			END_IF
		END_IF 
				
		(* CASE MAGAZINE LS MOVE *)
		IF NOT csp_case_feed_magazine_accU_lsDepth.in_position
		THEN
			case_feed_magazine_accU_lsDepth_move_req := TRUE;
		ELSE
			IF 	axis_is_disabled(csp_case_feed_magazine_accU_lsDepth.axis)
				AND csp_case_feed_magazine_accU_lsDepth.fsm_status = CSP_CASE_FEED_MAGAZINE_ACCU_LSDEPTH_STATUS_DISABLED
			THEN
				case_feed_magazine_accU_lsDepth_move_req := FALSE;
			END_IF
		END_IF
				
		(* CASE MAGAZINE OS MOVE *)
		IF NOT csp_case_feed_magazine_accU_osDepth.in_position
		THEN
			case_feed_magazine_accU_osDepth_move_req := TRUE;
		ELSE
			IF axis_is_disabled(csp_case_feed_magazine_accU_osDepth.axis)
			THEN
				case_feed_magazine_accU_osDepth_move_req := FALSE;
			END_IF
		END_IF
				
		(* TRANSPORT VM MOVE *)
		IF NOT csp_case_transport_accU_depth.in_position
		THEN
			case_transport_accU_depth_move_req := TRUE;
		END_IF
		
		IF 	csp_case_transport_accU_depth.in_position
			AND csp_case_feed_shuttle_accU_depth.in_position
		THEN
			case_transport_accU_depth_move_req := FALSE;
		END_IF
				
		(* ALL GROUP 1 NOT IN MOVE REQUEST - ADVANCE *)
		IF 	NOT transfer_accumulator_accU_depth_move_req
			AND NOT transfer_infeed_accU_depth_move_req
			AND NOT case_feed_magazine_accU_lsDepth_move_req
			AND NOT case_feed_magazine_accU_osDepth_move_req
			AND NOT case_transport_accU_depth_move_req
		THEN
			IF csp_case_tr_accU_ls_width.axis.actual_position < csp_case_tr_accU_ls_width.position_req
			THEN
				fsm_next_status := CSP_MAIN_ACCUCHANGE_STATUS_GROUP_2_TR_UP_ACCU_MOVE_REQUEST;
			ELSE
				fsm_next_status := CSP_MAIN_ACCUCHANGE_STATUS_GROUP_2_TR_DOWN_ACCU_MOVE_REQUEST;
			END_IF
		END_IF
		
	(*Top rail moves up, must move top rail before loader guides and glue guns to avoid conflict*)	
	CSP_MAIN_ACCUCHANGE_STATUS_GROUP_2_TR_UP_ACCU_MOVE_REQUEST:	
		
		(* TOP RAIL VM MOVE *)
		IF 	NOT csp_case_tr_accU_ls_width.in_position
			AND NOT csp_case_tr_accU_os_width.in_position
		THEN
			case_tr_accU_ls_width_move_req := TRUE;
		END_IF
		
		IF 	csp_case_tr_accU_ls_width.in_position
			AND csp_case_tr_accU_os_width.in_position
		THEN
			case_tr_accU_ls_width_move_req := FALSE;
			
			(* LS UPPER GLUE GUNS *)
			IF NOT csp_case_glue_ls_accu_upperposition.in_position
			THEN
				case_glue_ls_accU_upperPosition_move_req := TRUE;
			ELSE
				IF axis_is_disabled(csp_case_glue_ls_accu_upperposition.axis)
				THEN
					case_glue_ls_accU_upperPosition_move_req := FALSE;
				END_IF
				
				(* LS LOWER GLUE GUNS *)
				IF NOT csp_case_glue_ls_accu_lowerposition.in_position
				THEN
					case_glue_ls_accU_lowerPosition_move_req := TRUE;
				ELSE
					IF axis_is_disabled(csp_case_glue_ls_accu_lowerposition.axis)
					THEN
						case_glue_ls_accU_lowerPosition_move_req := FALSE;
					END_IF
				END_IF
			END_IF
			
			(* OS UPPER GLUE GUNS *)
			IF NOT csp_case_glue_os_accu_upperposition.in_position
			THEN
				case_glue_os_accU_upperPosition_move_req := TRUE;
			ELSE
				IF axis_is_disabled(csp_case_glue_os_accu_upperposition.axis)
				THEN
					case_glue_os_accU_upperPosition_move_req := FALSE;
				END_IF
				
				(* OS LOWER GLUE GUNS *)
				IF NOT csp_case_glue_os_accu_lowerposition.in_position
				THEN
					case_glue_os_accU_lowerPosition_move_req := TRUE;
				ELSE
					IF axis_is_disabled(csp_case_glue_os_accu_lowerposition.axis)
					THEN
						case_glue_os_accU_lowerPosition_move_req := FALSE;
					END_IF
				END_IF
			END_IF
			
			(* OS WIDTH GLUE *)
			IF NOT csp_case_glue_os_accu_width.in_position
			THEN
				case_glue_os_accU_width_move_req := TRUE;
			ELSE
				IF axis_is_disabled(csp_case_glue_os_accu_width.axis)
				THEN
					case_glue_os_accU_width_move_req := FALSE;
				END_IF
			END_IF
			
			(* LOADER GUIDE WIDTH MOVE *)
			IF NOT csp_case_loader_guide_accU_width.in_position
			THEN
				case_loader_guide_accU_width_move_req := TRUE;
			ELSE
				IF axis_is_disabled(csp_case_loader_guide_accU_width.axis)
				THEN
					case_loader_guide_accU_width_move_req := FALSE;
				END_IF
			END_IF
		
		
			(* TOP RAIL DEPTH = WAITS ON TOP RAIL WIDTH TO BE DONE *)
			IF NOT csp_case_tr_accu_depth.in_position
				AND NOT case_tr_accU_ls_width_move_req (* VERIFIES TOP RAIL WIDTH IS COMPLETED FIRST *)
			THEN
				case_tr_accU_depth_move_req := TRUE;
			ELSE
				IF axis_is_disabled(csp_case_tr_accu_depth.axis)
				THEN
					case_tr_accU_depth_move_req := FALSE;
				END_IF
			END_IF
		END_IF
		
		(* INFEED WATERFALL MOVE *)
		IF NOT csp_transfer_infeed_accU_waterfallAdjust.in_position
		THEN
			transfer_infeed_accU_waterfall_move_req := TRUE;
		ELSE
			IF 	axis_is_disabled(csp_transfer_infeed_accU_waterfallAdjust.axis)
				AND csp_transfer_infeed_accU_waterfallAdjust.fsm_status = CSP_TRANSFER_INFEED_ACCU_WATERFALL_ADJUST_STATUS_DISABLED
			THEN
				transfer_infeed_accU_waterfall_move_req := FALSE;
			END_IF
		END_IF
		
		(* ALL GROUP 2 NOT IN MOVE REQUEST - ADVANCE *)
		IF NOT case_tr_accU_ls_width_move_req
			AND NOT transfer_infeed_accU_waterfall_move_req
			AND NOT case_glue_ls_accU_lowerPosition_move_req
			AND NOT case_glue_ls_accU_upperPosition_move_req
			AND NOT case_glue_os_accU_lowerPosition_move_req
			AND NOT case_glue_os_accU_upperPosition_move_req
			AND NOT case_glue_os_accU_width_move_req
			AND NOT case_loader_guide_accU_width_move_req
			AND NOT case_tr_accU_depth_move_req
		THEN
			fsm_next_status := CSP_MAIN_ACCUCHANGE_STATUS_ADD_CASE_BLANKS;
		END_IF
		
	(*Top rail moves down, must move top rail after loader guides and glue guns to avoid conflict*)	
	CSP_MAIN_ACCUCHANGE_STATUS_GROUP_2_TR_DOWN_ACCU_MOVE_REQUEST:
		
		(* LS LOWER GLUE GUNS *)
		IF NOT csp_case_glue_ls_accu_lowerposition.in_position
		THEN
			case_glue_ls_accU_lowerPosition_move_req := TRUE;
		ELSE
			IF axis_is_disabled(csp_case_glue_ls_accu_lowerposition.axis)
			THEN
				case_glue_ls_accU_lowerPosition_move_req := FALSE;
			END_IF
		
		(* LS UPPER GLUE GUNS *)
			IF NOT csp_case_glue_ls_accu_upperposition.in_position
			THEN
				case_glue_ls_accU_upperPosition_move_req := TRUE;
			ELSE
				IF axis_is_disabled(csp_case_glue_ls_accu_upperposition.axis)
				THEN
					case_glue_ls_accU_upperPosition_move_req := FALSE;
				END_IF
			END_IF
			
			(* LOADER GUIDE WIDTH MOVE *)
			IF NOT csp_case_loader_guide_accU_width.in_position
			THEN
				case_loader_guide_accU_width_move_req := TRUE;
			ELSE
				IF axis_is_disabled(csp_case_loader_guide_accU_width.axis)
				THEN
					case_loader_guide_accU_width_move_req := FALSE;
				END_IF
			END_IF
		END_IF
		
		(* OS LOWER GLUE GUNS *)
		IF NOT csp_case_glue_os_accu_lowerposition.in_position
		THEN
			case_glue_os_accU_lowerPosition_move_req := TRUE;
		ELSE
			IF axis_is_disabled(csp_case_glue_os_accu_lowerposition.axis)
			THEN
				case_glue_os_accU_lowerPosition_move_req := FALSE;
			END_IF
		
		(* OS UPPER GLUE GUNS *)
			IF NOT csp_case_glue_os_accu_upperposition.in_position
			THEN
				case_glue_os_accU_upperPosition_move_req := TRUE;
			ELSE
				IF axis_is_disabled(csp_case_glue_os_accu_upperposition.axis)
				THEN
					case_glue_os_accU_upperPosition_move_req := FALSE;
				END_IF
			END_IF
		
		(* OS WIDTH GLUE *)
			IF NOT csp_case_glue_os_accu_width.in_position
			THEN
				case_glue_os_accU_width_move_req := TRUE;
			ELSE
				IF axis_is_disabled(csp_case_glue_os_accu_width.axis)
				THEN
					case_glue_os_accU_width_move_req := FALSE;
				END_IF
			END_IF
		END_IF
		
		(* TOP RAIL VM MOVE *)
		IF 	csp_case_glue_os_accu_upperposition.in_position
			AND csp_case_glue_ls_accu_upperposition.in_position
			AND csp_case_loader_guide_accU_width.in_position
			AND csp_case_glue_os_accu_width.in_position
			AND NOT csp_case_tr_accU_ls_width.in_position
			AND NOT csp_case_tr_accU_os_width.in_position
		THEN
			case_tr_accU_ls_width_move_req := TRUE;
		END_IF
		
		IF 	csp_case_tr_accU_ls_width.in_position
			AND csp_case_tr_accU_os_width.in_position
		THEN
			case_tr_accU_ls_width_move_req := FALSE;
		
			(* TOP RAIL DEPTH = WAITS ON TOP RAIL WIDTH TO BE DONE *)
			IF NOT csp_case_tr_accu_depth.in_position
			THEN
				case_tr_accU_depth_move_req := TRUE;
			ELSE
				IF axis_is_disabled(csp_case_tr_accu_depth.axis)
				THEN
					case_tr_accU_depth_move_req := FALSE;
				END_IF
			END_IF
		END_IF		
		
		(* INFEED WATERFALL MOVE *)
		IF NOT csp_transfer_infeed_accU_waterfallAdjust.in_position
		THEN
			transfer_infeed_accU_waterfall_move_req := TRUE;
		ELSE
			IF 	axis_is_disabled(csp_transfer_infeed_accU_waterfallAdjust.axis)
				AND csp_transfer_infeed_accU_waterfallAdjust.fsm_status = CSP_TRANSFER_INFEED_ACCU_WATERFALL_ADJUST_STATUS_DISABLED
			THEN
				transfer_infeed_accU_waterfall_move_req := FALSE;
			END_IF
		END_IF
		
		(* ALL GROUP 2 NOT IN MOVE REQUEST - ADVANCE *)
		IF 	NOT case_tr_accU_ls_width_move_req
			AND NOT transfer_infeed_accU_waterfall_move_req
			AND NOT case_glue_ls_accU_lowerPosition_move_req
			AND NOT case_glue_ls_accU_upperPosition_move_req
			AND NOT case_glue_os_accU_lowerPosition_move_req
			AND NOT case_glue_os_accU_upperPosition_move_req
			AND NOT case_glue_os_accU_width_move_req
			AND NOT case_loader_guide_accU_width_move_req
			AND NOT case_tr_accU_depth_move_req
		THEN
			fsm_next_status := CSP_MAIN_ACCUCHANGE_STATUS_ADD_CASE_BLANKS;
		END_IF
		
		
	CSP_MAIN_ACCUCHANGE_STATUS_ADD_CASE_BLANKS:
	
		hmi_current_accU_step := 7; //"Add Case Blanks to Magazine"
		
		IF 
			(
				csp_main.is_SFI
				AND csp_case_feed_magazine_level.level_status <= csp_case_feed_magazine_level.LEVEL_STATUS_LOW_LEVEL
			)
			OR
			(
				NOT csp_main.is_SFI
				AND csp_case_feed_magazine_level.level_status >= csp_case_feed_magazine_level.LEVEL_STATUS_MIN_LEVEL
			)		
		THEN
			navigate_to_accU_popup := FALSE;
			Motion_Motors_New_Size_Req := TRUE;
			hmi_current_accU_step := 0;
			machine_size_complete := TRUE;
			Brand_Change_Occurred := FALSE;
			fsm_next_status := CSP_MAIN_ACCUCHANGE_STATUS_BRAND_CHECK;
		END_IF
		
END_CASE;


(* ADVANCES TO NEXT STEP *)
IF 	NOT debug_fsm
	OR
	debug_fsm_one_step	
THEN
	fsm_status := fsm_next_status;
	debug_fsm_one_step := FALSE;
END_IF


(* Connection timeout *)
IF	fsm_running
	AND NOT debug_fsm
THEN
	IF	timer_is_expired(fsm_tmr)
	THEN
		process_message_set(1, fsm_status, 0, changeover_timeout_asm);
	END_IF
ELSE
	timer_restart(600000, fsm_tmr);
END_IF



(* CHECKS ALL RFID TAGS BEFORE RUNNING IF APPLICABLE *)
motorization_conditioner_start_done(eoat_rfid_checked_motcond);
motorization_conditioner_start_done(loader_pusher_rfid_checked_motcond);
motorization_conditioner_start_done(loader_plate_rfid_checked_motcond);

CASE running_rfid_status OF	
	READ_RUNNING_CHECK_STATUS_START:
	
		rfid_read_write_running := TRUE;
		running_rfid_status_next := READ_RUNNING_CHECK_STATUS_EOAT_CHECK_CP;
		
	(* EOAT CHECK *)
	READ_RUNNING_CHECK_STATUS_EOAT_CHECK_CP:
	
		IF csp_case_feed_virtualMaster.phase_done
		THEN
			IF csp_case_feed_arm_sensors.rfid_input_bitheader_1.CP
				AND csp_case_feed_arm_sensors.rfid_input_bitheader_2.CP
			THEN
				RFID_reader_list_accuchange := CASE_FEED_EOAT_READER;
				running_rfid_status_next := READ_RUNNING_CHECK_STATUS_EOAT_SEND_READ;
			ELSE
				motorization_conditioner_start_done(eoat_rfid_checked_motcond);
				running_rfid_status_next := READ_RUNNING_CHECK_STATUS_LOADER_PUSHER_CHECK_CP;
			END_IF
		END_IF
		
		
	READ_RUNNING_CHECK_STATUS_EOAT_SEND_READ:
	
		RFID_reading := TRUE;
		
		IF csp_case_feed_arm_sensors.rfid_read_done
		THEN
			running_rfid_status_next := READ_RUNNING_CHECK_STATUS_EOAT_CHECK_READ;
		END_IF
		
		
	READ_RUNNING_CHECK_STATUS_EOAT_CHECK_READ:
	
		RFID_reading := FALSE;
		
		IF csp_case_feed_arm_sensors.rfid_value = INT_TO_BYTE(hmi_change_part_eoat_color)
		THEN
			motorization_conditioner_start_done(eoat_rfid_checked_motcond);
			running_rfid_status_next := READ_RUNNING_CHECK_STATUS_LOADER_PUSHER_CHECK_CP;
		ELSE
			process_message_set(1, 1, 1, change_part_eoat_wrong);
		END_IF
		
		
	(* LOADER PUSHER CHECK *)
	READ_RUNNING_CHECK_STATUS_LOADER_PUSHER_CHECK_CP:
		
		IF axis_is_cam_engaged(csp_case_loader_pusher.axis)
		THEN
			IF csp_case_loader_pusher.rfid_input_bitheader_1.CP
				AND csp_case_loader_pusher.rfid_input_bitheader_2.CP
			THEN
				RFID_reader_list_accuchange := LOADER_PUSHER_READER;
				running_rfid_status_next := READ_RUNNING_CHECK_STATUS_LOADER_PUSHER_SEND_READ;
			ELSE
				motorization_conditioner_start_done(loader_pusher_rfid_checked_motcond);
				running_rfid_status_next := READ_RUNNING_CHECK_STATUS_LOADER_PLATE_CHECK_CP;
			END_IF
		END_IF
			
		
	READ_RUNNING_CHECK_STATUS_LOADER_PUSHER_SEND_READ:
	
		RFID_reading := TRUE;
		
		IF csp_case_loader_pusher.rfid_read_done
		THEN
			running_rfid_status_next := READ_RUNNING_CHECK_STATUS_LOADER_PUSHER_CHECK_READ;
		END_IF

		
	READ_RUNNING_CHECK_STATUS_LOADER_PUSHER_CHECK_READ:
	
		RFID_reading := FALSE;
		
		IF csp_case_loader_pusher.rfid_value = INT_TO_BYTE(hmi_change_part_pusher_color)
		THEN
			motorization_conditioner_start_done(loader_pusher_rfid_checked_motcond);
			running_rfid_status_next := READ_RUNNING_CHECK_STATUS_LOADER_PLATE_CHECK_CP;
		ELSE
			process_message_set(1, 1, 1, change_part_pusher_wrong);
		END_IF
		
		
	(* LOADER PLATE CHECK *)
	READ_RUNNING_CHECK_STATUS_LOADER_PLATE_CHECK_CP:
	
		IF 	csp_case_loader_sensors.rfid_input_bitheader_1.CP
			AND csp_case_loader_sensors.rfid_input_bitheader_2.CP
		THEN
			RFID_reader_list_accuchange := LOADER_GUIDE_PLATE_READER;
			running_rfid_status_next := READ_RUNNING_CHECK_STATUS_LOADER_PUSHER_SEND_READ;
		ELSE
			motorization_conditioner_start_done(loader_plate_rfid_checked_motcond);
			running_rfid_status_next := READ_RUNNING_CHECK_STATUS_LOADER_PLATE_CHECK_CP;
		END_IF
		
		
	READ_RUNNING_CHECK_STATUS_LOADER_PLATE_SEND_READ:
		
		RFID_reading := TRUE;
		
		IF csp_case_loader_sensors.rfid_read_done
		THEN
			running_rfid_status_next := READ_RUNNING_CHECK_STATUS_LOADER_PLATE_CHECK_READ;
		END_IF
		
		
	READ_RUNNING_CHECK_STATUS_LOADER_PLATE_CHECK_READ:
	
		RFID_reading := FALSE;
		
		IF csp_case_loader_sensors.rfid_value = INT_TO_BYTE(hmi_change_part_plate_color)
		THEN
			motorization_conditioner_start_done(loader_plate_rfid_checked_motcond);
			running_rfid_status_next := READ_RUNNING_CHECK_STATUS_DONE;
		ELSE
			process_message_set(1, 1, 1, change_part_plate_wrong);
		END_IF
		
	(* ALL CHECKED *)
	READ_RUNNING_CHECK_STATUS_DONE:
	
		rfid_read_write_running := FALSE;
		
		IF axis_is_moving(csp_main_motorization_virtualManager.axis)
		THEN
			running_rfid_status_next := READ_RUNNING_CHECK_STATUS_WAITING;
		END_IF
		
		
	READ_RUNNING_CHECK_STATUS_WAITING:
		
		;
		
		
	READ_RUNNING_CHECK_STATUS_ERROR:
	
		;
		
		
END_CASE

running_rfid_status := running_rfid_status_next;

IF 	machine_is_stopped(csp.mch)
	OR machine_is_stop_emergency_active(csp.mch)
THEN
	process_message_reset(change_part_eoat_wrong);
	process_message_reset(change_part_pusher_wrong);
	process_message_reset(change_part_plate_wrong);
END_IF


(************************************************************************)


(* HORN CONTROL FOR ANY ACC-U-CHANGE MOTOR MOVING *)
IF (
		axis_is_moving(csp_case_transport_accU_depth.axis)
		AND 
		NOT axis_is_disabled(csp_case_transport_accU_depth.axis)
	)
	OR	
	(
		axis_is_moving(csp_case_feed_shuttle_accU_depth.axis)
		AND 
		NOT axis_is_disabled(csp_case_feed_shuttle_accU_depth.axis)
	)
	OR	
	(
		axis_is_moving(csp_case_feed_magazine_accU_lsDepth.axis)
		AND 
		NOT axis_is_disabled(csp_case_feed_magazine_accU_lsDepth.axis)
	)
	OR
	(
		axis_is_moving(csp_case_feed_magazine_accU_osDepth.axis)
		AND 
		NOT axis_is_disabled(csp_case_feed_magazine_accU_osDepth.axis)
	)
	OR
	(
		axis_is_moving(csp_case_feed_reject_accU_depth.axis)
		AND 
		NOT axis_is_disabled(csp_case_feed_reject_accU_depth.axis)
	)
	OR
	(
		axis_is_moving(csp_transfer_infeed_accU_depth.axis)
		AND 
		NOT axis_is_disabled(csp_transfer_infeed_accU_depth.axis)
	)
	OR
	(
		axis_is_moving(csp_transfer_accumulator_accU_depth.axis)
		AND 
		NOT axis_is_disabled(csp_transfer_accumulator_accU_depth.axis)
	)
	OR
	(
		axis_is_moving(csp_transfer_infeed_accU_waterfallAdjust.axis)
		AND 
		NOT axis_is_disabled(csp_transfer_infeed_accU_waterfallAdjust.axis)
	)
	OR
	(
		axis_is_moving(csp_transfer_accumulator_accU_convDepth.axis)
		AND 
		NOT axis_is_disabled(csp_transfer_accumulator_accU_convDepth.axis)
	)
	OR
	(
		axis_is_moving(csp_case_tr_accU_depth.axis)
		AND 
		NOT axis_is_disabled(csp_case_tr_accU_depth.axis)
	)
	OR
	(
		axis_is_moving(csp_case_loader_guide_accU_width.axis)
		AND 
		NOT axis_is_disabled(csp_case_loader_guide_accU_width.axis)
	)
	OR
	(
		axis_is_moving(csp_case_glue_os_accU_width.axis)
		AND 
		NOT axis_is_disabled(csp_case_glue_os_accU_width.axis)
	)
	OR
	(
		axis_is_moving(csp_case_glue_os_accU_upperPosition.axis)
		AND 
		NOT axis_is_disabled(csp_case_glue_os_accU_upperPosition.axis)
	)
	OR
	(
		axis_is_moving(csp_case_glue_os_accU_lowerPosition.axis)
		AND 
		NOT axis_is_disabled(csp_case_glue_os_accU_lowerPosition.axis)
	)
	OR
	(
		axis_is_moving(csp_case_glue_ls_accU_upperPosition.axis)
		AND 
		NOT axis_is_disabled(csp_case_glue_ls_accU_upperPosition.axis)
	)
	OR
	(
		axis_is_moving(csp_case_glue_ls_accU_lowerPosition.axis)
		AND 
		NOT axis_is_disabled(csp_case_glue_ls_accU_lowerPosition.axis)
	)
	OR
	(
		axis_is_moving(csp_case_tr_accU_os_width.axis)
		AND 
		NOT axis_is_disabled(csp_case_tr_accU_os_width.axis)
	)
	OR
	(
		axis_is_moving(csp_case_tr_accU_ls_width.axis)
		AND 
		NOT axis_is_disabled(csp_case_tr_accU_ls_width.axis)
	)
THEN
	accU_axis_moving := TRUE;
ELSE
	accU_axis_moving := FALSE;
END_IF


IF 	accU_axis_moving
	AND filter_is_off(horn_on_filter)
THEN
	accU_axis_moving_horn_on := TRUE;
END_IF

IF filter_is_on(horn_on_filter)
THEN
	accU_axis_moving_horn_on := FALSE;
END_IF


filter_set_delays(
	delay_off_on			:= horn_on_time,
	delay_on_off			:= horn_off_time,
	CONVERSION_this			:= horn_on_filter);

//Added to prevent the move request from staying ON and alway moving to the phase position
IF 	csp_main_accuchange.hmi_brand_status_color_hgos.status = HMI_OBJECT_STATUS_ON
THEN
	case_transport_accU_depth_move_req := FALSE; 
	case_feed_magazine_accU_lsDepth_move_req := FALSE; 
	case_feed_magazine_accU_osDepth_move_req := FALSE;
	transfer_infeed_accU_depth_move_req := FALSE;
	transfer_infeed_accU_waterfall_move_req := FALSE;
	transfer_accumulator_accU_depth_move_req:= FALSE; 
	case_tr_accU_depth_move_req := FALSE;
	case_loader_guide_accU_width_move_req := FALSE;
	case_glue_os_accU_width_move_req := FALSE;
	case_glue_os_accU_upperPosition_move_req := FALSE;
	case_glue_os_accU_lowerPosition_move_req := FALSE;
	case_glue_ls_accU_upperPosition_move_req := FALSE;
	case_glue_ls_accU_lowerPosition_move_req := FALSE;
	case_tr_accU_ls_width_move_req:= FALSE; 
END_IF



_handle_messages();

_write_output();


IF NOT first_scan_bool
THEN
	cam_data_changed := TRUE;
	not_in_brand_change := TRUE;
END_IF

IF first_scan_bool
	AND cam_data_changed
	AND NOT Brand_Change_Occurred
THEN
	cam_data_changed := FALSE;
END_IF


first_scan_bool := TRUE;

